  gc_DbmTranslation_fr_Text97 : WSTRING(28) := "White Light AVG actual value";
  gc_DbmTranslation_fr_Text98 : WSTRING(23) := "White Light AVD command";
  gc_DbmTranslation_fr_Text99 : WSTRING(28) := "White Light AVD actual value";
  gc_DbmTranslation_fr_Text100 : WSTRING(21) := "Red Light AVG command";
  gc_DbmTranslation_fr_Text101 : WSTRING(26) := "Red Light AVG actual value";
  gc_DbmTranslation_fr_Text102 : WSTRING(21) := "Red Light AVD command";
  gc_DbmTranslation_fr_Text103 : WSTRING(26) := "Red Light AVD actual value";
  gc_DbmTranslation_fr_Text104 : WSTRING(23) := "White Light ARG command";
  gc_DbmTranslation_fr_Text105 : WSTRING(28) := "White Light ARG actual value";
  gc_DbmTranslation_fr_Text106 : WSTRING(23) := "White Light ARD command";
  gc_DbmTranslation_fr_Text107 : WSTRING(28) := "White Light ARD actual value";
  gc_DbmTranslation_fr_Text108 : WSTRING(21) := "Red Light ARG command";
  gc_DbmTranslation_fr_Text109 : WSTRING(26) := "Red Light ARG actual value";
  gc_DbmTranslation_fr_Text110 : WSTRING(21) := "Red Light ARD command";
  gc_DbmTranslation_fr_Text111 : WSTRING(26) := "Red Light ARD actual value";
  gc_DbmTranslation_fr_Text112 : WSTRING(29) := "Suplly Pvg Left Track command";
  gc_DbmTranslation_fr_Text113 : WSTRING(34) := "Suplly Pvg Left Track actual value";
  gc_DbmTranslation_fr_Text114 : WSTRING(30) := "Suplly Pvg Right Track command";
  gc_DbmTranslation_fr_Text115 : WSTRING(35) := "Suplly Pvg Right Track actual value";
  gc_DbmTranslation_fr_Text116 : WSTRING(33) := "Ev UnBlock Oscillation Axle state";
  gc_DbmTranslation_fr_Text117 : WSTRING(40) := "Ev UnBlock Oscillation Axle command bool";
  gc_DbmTranslation_fr_Text118 : WSTRING(26) := "Ev Up Axle Oscillant state";
  gc_DbmTranslation_fr_Text119 : WSTRING(33) := "Ev Up Axle Oscillant Command Bool";
  gc_DbmTranslation_fr_Text120 : WSTRING(29) := "Ev Down Axle Oscillant  state";
  gc_DbmTranslation_fr_Text121 : WSTRING(35) := "Ev Down Axle Oscillant Command Bool";
  gc_DbmTranslation_fr_Text122 : WSTRING(20) := "Ev Up AxleFixe state";
  gc_DbmTranslation_fr_Text123 : WSTRING(28) := "Ev Up Axle Fixe Command Bool";
  gc_DbmTranslation_fr_Text124 : WSTRING(22) := "Ev Down AxleFixe state";
  gc_DbmTranslation_fr_Text125 : WSTRING(30) := "Ev Down Axle Fixe Command Bool";
  gc_DbmTranslation_fr_Text126 : WSTRING(35) := "Ev Park Brake Axle Oscillant  state";
  gc_DbmTranslation_fr_Text127 : WSTRING(42) := "Ev Park Brake Axle Oscillant  command bool";
  gc_DbmTranslation_fr_Text128 : WSTRING(29) := "Ev Park Brake Axle Fixe state";
  gc_DbmTranslation_fr_Text129 : WSTRING(37) := "Ev Park Brake Axle Fixe  command bool";
  gc_DbmTranslation_fr_Text130 : WSTRING(37) := "Ev Service Brake Axle Oscillant state";
  gc_DbmTranslation_fr_Text131 : WSTRING(36) := "Ev Service Brake Axle 1 command Bool";
  gc_DbmTranslation_fr_Text132 : WSTRING(32) := "Ev Service Brake Axle Fixe state";
  gc_DbmTranslation_fr_Text133 : WSTRING(36) := "Ev Service Brake Axle 2 command Bool";
  gc_DbmTranslation_fr_Text134 : WSTRING(19) := "Klaxon Neotec state";
  gc_DbmTranslation_fr_Text135 : WSTRING(26) := "Klaxon Neotec command bool";
  gc_DbmTranslation_fr_Text136 : WSTRING(18) := "Forward pump state";
  gc_DbmTranslation_fr_Text137 : WSTRING(21) := "Forward pump  command";
  gc_DbmTranslation_fr_Text138 : WSTRING(27) := "Forward pump actual current";
  gc_DbmTranslation_fr_Text139 : WSTRING(19) := "Backward pump state";
  gc_DbmTranslation_fr_Text140 : WSTRING(22) := "Backward pump  command";
  gc_DbmTranslation_fr_Text141 : WSTRING(28) := "Backward pump actual current";
  gc_DbmTranslation_fr_Text142 : WSTRING(22) := "Pvg left track command";
  gc_DbmTranslation_fr_Text143 : WSTRING(29) := "Pvg left track actual voltage";
  gc_DbmTranslation_fr_Text144 : WSTRING(23) := "Pvg right track command";
  gc_DbmTranslation_fr_Text145 : WSTRING(30) := "Pvg right track actual voltage";
  gc_DbmTranslation_fr_Text146 : WSTRING(26) := "Supply Ana Sensors Command";
  gc_DbmTranslation_fr_Text147 : WSTRING(24) := "Supply Ana Sensors Value";
  gc_DbmTranslation_fr_Text148 : WSTRING(30) := "Pvg Left Track Lowside Command";
  gc_DbmTranslation_fr_Text149 : WSTRING(28) := "Pvg Left Track Lowside Value";
  gc_DbmTranslation_fr_Text150 : WSTRING(31) := "Pvg Right Track Lowside Command";
  gc_DbmTranslation_fr_Text151 : WSTRING(29) := "Pvg Right Track Lowside Value";
  gc_DbmTranslation_fr_Text152 : WSTRING(39) := "Return low side Ev Forward Pump command";
  gc_DbmTranslation_fr_Text153 : WSTRING(37) := "Return low side Ev Forward Pump state";
  gc_DbmTranslation_fr_Text154 : WSTRING(40) := "Return low side Ev Backward Pump command";
  gc_DbmTranslation_fr_Text155 : WSTRING(38) := "Return low side Ev Backward Pump state";
  gc_DbmTranslation_fr_Text156 : WSTRING(19) := "Neon Lights command";
  gc_DbmTranslation_fr_Text157 : WSTRING(17) := "Neon Lights value";
  gc_DbmTranslation_fr_Text158 : WSTRING(33) := "Ev 2 Deflector Transmission value";
  gc_DbmTranslation_fr_Text159 : WSTRING(21) := "Cooling relay command";
  gc_DbmTranslation_fr_Text160 : WSTRING(19) := "Cooling relay state";
  gc_DbmTranslation_fr_Text161 : WSTRING(54) := "Sorties d’activation de l’Ev du deuxième frein de parc";
  gc_DbmTranslation_fr_Text162 : WSTRING(54) := "Sorties d’activation de l’Ev du deuxième frein de parc";
  gc_DbmTranslation_fr_Text163 : WSTRING(33) := "Ev 2nd Park Brake Axle Fixe State";
  gc_DbmTranslation_fr_Text164 : WSTRING(33) := "Ev 2nd Park Brake Axle Osci State";
  gc_DbmTranslation_fr_Text165 : WSTRING(41) := "Pvg Translation for Rail Electric Command";
  gc_DbmTranslation_fr_Text166 : WSTRING(41) := "Pvg Translation for Rail Electric Voltage";
  gc_DbmTranslation_fr_Text167 : WSTRING(48) := "Suplly Pvg Translation for Rail Electric Command";
  gc_DbmTranslation_fr_Text168 : WSTRING(46) := "Suplly Pvg Translation for Rail Electric State";
  gc_DbmTranslation_fr_Text169 : WSTRING(42) := "Ev Deviator for Rail Electric Mode Command";
  gc_DbmTranslation_fr_Text170 : WSTRING(40) := "Ev Deviator for Rail Electric Mode State";
  gc_DbmTranslation_fr_Text171 : WSTRING(43) := "Relay Cut Off Variator for Electric Command";
  gc_DbmTranslation_fr_Text172 : WSTRING(41) := "Relay Cut Off Variator for Electric State";
  gc_DbmTranslation_fr_Text173 : WSTRING(28) := "Relay Enable Battery Command";
  gc_DbmTranslation_fr_Text174 : WSTRING(26) := "Relay Enable Battery State";
  gc_DbmTranslation_fr_Text175 : WSTRING(25) := "Byte increased each cycle";
  gc_DbmTranslation_fr_Text176 : WSTRING(22) := "Watchdog current state";
  gc_DbmTranslation_fr_Text177 : WSTRING(11) := "Ecu voltage";
  gc_DbmTranslation_fr_Text178 : WSTRING(13) := "Off Rail Mode";
  gc_DbmTranslation_fr_Text179 : WSTRING(9) := "Rail Mode";
  gc_DbmTranslation_fr_Text180 : WSTRING(75) := "Output value Lut of Manipulator left radio control in range -10000 to 10000";
  gc_DbmTranslation_fr_Text181 : WSTRING(35) := "Output value Lut of Left Track Pvg ";
  gc_DbmTranslation_fr_Text182 : WSTRING(76) := "Output value Lut of Manipulator Right radio control in range -10000 to 10000";
  gc_DbmTranslation_fr_Text183 : WSTRING(36) := "Output value Lut of Right Track Pvg ";
  gc_DbmTranslation_fr_Text184 : WSTRING(52) := "Outût value Lut of Joystick advance Rail translation";
  gc_DbmTranslation_fr_Text185 : WSTRING(40) := "Output Lut  of Forward Pump Transmission";
  gc_DbmTranslation_fr_Text186 : WSTRING(41) := "Output Lut  of Backward Pump Transmission";
  gc_DbmTranslation_fr_Text187 : WSTRING(71) := "Calculate consigne current of Forward Pump transmission on percent *100";
  gc_DbmTranslation_fr_Text188 : WSTRING(24) := "LastJoystickAdvanceValue";
  gc_DbmTranslation_fr_Text189 : WSTRING(37) := "Scaling Value of Joystick advancement";
  gc_DbmTranslation_fr_Text190 : WSTRING(39) := "State of service brake rail translation";
  gc_DbmTranslation_fr_Text191 : WSTRING(36) := "Enable Start timer for service brake";
  gc_DbmTranslation_fr_Text192 : WSTRING(48) := "Speed motor command provide by track transaltion";
  gc_DbmTranslation_fr_Text193 : WSTRING(28) := "Force silent mode motor test";
  gc_DbmTranslation_fr_Text194 : WSTRING(19) := "Angular sensor test";
  gc_DbmTranslation_fr_Text195 : WSTRING(17) := "Speed axle sensor";
  gc_DbmTranslation_fr_Text196 : WSTRING(18) := "Average Time cycle";
  gc_DbmTranslation_fr_Text197 : WSTRING(14) := "Max time cycle";
  gc_DbmTranslation_fr_Text198 : WSTRING(40) := "First translation for release park brake";
  gc_DbmTranslation_fr_Text199 : WSTRING(35) := "Autorize Up Axle Oscillant movement";
  gc_DbmTranslation_fr_Text200 : WSTRING(37) := "Autorize Down Axle Oscillant movement";
  gc_DbmTranslation_fr_Text201 : WSTRING(30) := "Autorize Up Axle fixe movement";
  gc_DbmTranslation_fr_Text202 : WSTRING(32) := "Autorize Down Axle fixe movement";
  gc_DbmTranslation_fr_Text203 : WSTRING(19) := "Engine On run phase";
  gc_DbmTranslation_fr_Text204 : WSTRING(74) := "Transaltion rail or off rail is solicited , flag send to C1 to pilot motor";
  gc_DbmTranslation_fr_Text205 : WSTRING(42) := "Direction of rail translation (Av Ar Stop)";
  gc_DbmTranslation_fr_Text206 : WSTRING(39) := "Set condition to active Aru radio alarm";
  gc_DbmTranslation_fr_Text207 : WSTRING(36) := "Joystick advance setpoint after ramp";
  gc_DbmTranslation_fr_Text208 : WSTRING(46) := "Stabilized stop flag to active park brake rail";
  gc_DbmTranslation_fr_Text209 : WSTRING(48) := "Emergency brake flag to active sequence of brake";
  gc_DbmTranslation_fr_Text210 : WSTRING(51) := "Flag when the timer emergency service brake is done";
  gc_DbmTranslation_fr_Text211 : WSTRING(66) := "Flag when the timer stopped machine unblock osciilant axle is done";
  gc_DbmTranslation_fr_Text212 : WSTRING(86) := "Output value Lut of Manipulator left radio control in range -10000 to 10000 after ramp";
  gc_DbmTranslation_fr_Text213 : WSTRING(87) := "Output value Lut of Manipulator right radio control in range -10000 to 10000 after ramp";
  gc_DbmTranslation_fr_Text214 : WSTRING(52) := "Delta beetwen left and right Pvg crawler advancement";
  gc_DbmTranslation_fr_Text215 : WSTRING(65) := "Consigne left pvg track calcul with delta beetween left and right";
  gc_DbmTranslation_fr_Text216 : WSTRING(66) := "Consigne right pvg track calcul with delta beetween left and right";
  gc_DbmTranslation_fr_Text217 : WSTRING(56) := "Flag to detect brake when gachette or pedal are released";
  gc_DbmTranslation_fr_Text218 : WSTRING(50) := "Counter for debug when alarm aru radio is detected";
  gc_DbmTranslation_fr_Text219 : WSTRING(28) := "Red light ARG basket command";
  gc_DbmTranslation_fr_Text220 : WSTRING(30) := "White light ARG basket command";
  gc_DbmTranslation_fr_Text221 : WSTRING(32) := "Portilon close and ladder folded";
  gc_DbmTranslation_fr_Text222 : WSTRING(46) := "Test boolean  command to refresh objet evision";
  gc_DbmTranslation_fr_Text223 : WSTRING(60) := "Position of joysstick advancment ( AV_JOY, NEU_JOY , AR_JOY)";
  gc_DbmTranslation_fr_Text224 : WSTRING(81) := "Retain position of joystick advancement , reset when brake sequence is sollicited";
  gc_DbmTranslation_fr_Text225 : WSTRING(37) := "Authorize forward crawler translation";
  gc_DbmTranslation_fr_Text226 : WSTRING(38) := "Authorize backward crawler translation";
  gc_DbmTranslation_fr_Text227 : WSTRING(22) := "Return value uart init";
  gc_DbmTranslation_fr_Text228 : WSTRING(35) := "Authorize translation rail movement";
  gc_DbmTranslation_fr_Text229 : WSTRING(25) := "Ev forward track consigne";
  gc_DbmTranslation_fr_Text230 : WSTRING(24) := "Ev forward rail consigne";
  gc_DbmTranslation_fr_Text231 : WSTRING(0) := "";
  gc_DbmTranslation_fr_Text232 : WSTRING(21) := "Variable debug Neotec";
  gc_DbmTranslation_fr_Text233 : WSTRING(21) := "Variable debug Neotec";
  gc_DbmTranslation_fr_Text234 : WSTRING(21) := "Variable debug Neotec";
  gc_DbmTranslation_fr_Text235 : WSTRING(21) := "Variable debug Neotec";
  gc_DbmTranslation_fr_Text236 : WSTRING(21) := "Variable debug Neotec";
  gc_DbmTranslation_fr_Text237 : WSTRING(21) := "Variable debug Neotec";
  gc_DbmTranslation_fr_Text238 : WSTRING(21) := "Variable debug Neotec";
  gc_DbmTranslation_fr_Text239 : WSTRING(21) := "Variable debug Neotec";
  gc_DbmTranslation_fr_Text240 : WSTRING(21) := "Variable debug Neotec";
  gc_DbmTranslation_fr_Text241 : WSTRING(21) := "Variable debug Neotec";
  gc_DbmTranslation_fr_Text242 : WSTRING(21) := "Variable debug Neotec";
  gc_DbmTranslation_fr_Text243 : WSTRING(21) := "Variable debug Neotec";
  gc_DbmTranslation_fr_Text244 : WSTRING(21) := "Variable debug Neotec";
  gc_DbmTranslation_fr_Text245 : WSTRING(21) := "Variable debug Neotec";
  gc_DbmTranslation_fr_Text246 : WSTRING(21) := "Variable debug Neotec";
  gc_DbmTranslation_fr_Text247 : WSTRING(21) := "Variable debug Neotec";
  gc_DbmTranslation_fr_Text248 : WSTRING(21) := "Variable debug Neotec";
  gc_DbmTranslation_fr_Text249 : WSTRING(21) := "Variable debug Neotec";
  gc_DbmTranslation_fr_Text250 : WSTRING(21) := "Variable debug Neotec";
  gc_DbmTranslation_fr_Text251 : WSTRING(21) := "Variable debug Neotec";
  gc_DbmTranslation_fr_Text252 : WSTRING(21) := "Variable debug Neotec";
  gc_DbmTranslation_fr_Text253 : WSTRING(21) := "Variable debug Neotec";
  gc_DbmTranslation_fr_Text254 : WSTRING(21) := "Variable debug Neotec";
  gc_DbmTranslation_fr_Text255 : WSTRING(21) := "Variable debug Neotec";
  gc_DbmTranslation_fr_Text256 : WSTRING(21) := "Variable debug Neotec";
  gc_DbmTranslation_fr_Text257 : WSTRING(21) := "Variable debug Neotec";
  gc_DbmTranslation_fr_Text258 : WSTRING(21) := "Variable debug Neotec";
  gc_DbmTranslation_fr_Text259 : WSTRING(21) := "Variable debug Neotec";
  gc_DbmTranslation_fr_Text260 : WSTRING(21) := "Variable debug Neotec";
  gc_DbmTranslation_fr_Text261 : WSTRING(21) := "Variable debug Neotec";
  gc_DbmTranslation_fr_Text262 : WSTRING(21) := "Variable debug Neotec";
  gc_DbmTranslation_fr_Text263 : WSTRING(21) := "Variable debug Neotec";
  gc_DbmTranslation_fr_Text264 : WSTRING(21) := "Variable debug Neotec";
  gc_DbmTranslation_fr_Text265 : WSTRING(21) := "Variable debug Neotec";
  gc_DbmTranslation_fr_Text266 : WSTRING(21) := "Variable debug Neotec";
  gc_DbmTranslation_fr_Text267 : WSTRING(21) := "Variable debug Neotec";
  gc_DbmTranslation_fr_Text268 : WSTRING(21) := "Variable debug Neotec";
  gc_DbmTranslation_fr_Text269 : WSTRING(21) := "Variable debug Neotec";
  gc_DbmTranslation_fr_Text270 : WSTRING(21) := "Variable debug Neotec";
  gc_DbmTranslation_fr_Text271 : WSTRING(21) := "Variable debug Neotec";
  gc_DbmTranslation_fr_Text272 : WSTRING(28) := "Red light ARD basket command";
  gc_DbmTranslation_fr_Text273 : WSTRING(30) := "White light ARD basket command";
  gc_DbmTranslation_fr_Text274 : WSTRING(26) := "Active failure is detected";
  gc_DbmTranslation_fr_Text275 : WSTRING(19) := "Reduction pump rail";
  gc_DbmTranslation_fr_Text276 : WSTRING(20) := "Reduction pump track";
  gc_DbmTranslation_fr_Text277 : WSTRING(25) := "Active white lights 15746";
  gc_DbmTranslation_fr_Text278 : WSTRING(24) := "White light Av 15746 Cmd";
  gc_DbmTranslation_fr_Text279 : WSTRING(24) := "White light Ar 15746 Cmd";
  gc_DbmTranslation_fr_Text280 : WSTRING(38) := "Shunt all logic to test electricall IO";
  gc_DbmTranslation_fr_Text281 : WSTRING(29) := "Send Event Datalogger Message";
  gc_DbmTranslation_fr_Text282 : WSTRING(21) := "Depend de l’option MG";
  gc_DbmTranslation_fr_Text283 : WSTRING(13) := "Slow Blinking";
  gc_DbmTranslation_fr_Text284 : WSTRING(14) := "Total distance";
  gc_DbmTranslation_fr_Text285 : WSTRING(19) := "Running Stable 48XS";
  gc_DbmTranslation_fr_Text286 : WSTRING(39) := "Alarm Hydraulic Temperature Rail Active";
  gc_DbmTranslation_fr_Text287 : WSTRING(42) := "Alarm Hydraulic Temperature Crawler Active";
  gc_DbmTranslation_fr_Text288 : WSTRING(17) := "Diag Faulty Value";
  gc_DbmTranslation_fr_Text289 : WSTRING(15) := "Diag Device Num";
  gc_DbmTranslation_fr_Text290 : WSTRING(15) := "Diag Error Code";
  gc_DbmTranslation_fr_Text291 : WSTRING(21) := "Engine running stable";
  gc_DbmTranslation_fr_Text292 : WSTRING(42) := "Select config hollandaise to control light";
  gc_DbmTranslation_fr_Text293 : WSTRING(37) := "Portillon is installed on the machine";
  gc_DbmTranslation_fr_Text294 : WSTRING(34) := "Ladder is installed on the machine";
  gc_DbmTranslation_fr_Text295 : WSTRING(41) := "Measuring mat is installed on the machine";
  gc_DbmTranslation_fr_Text296 : WSTRING(107) := "-SpeedMaxRail Acces Site- Inclinaison Baslet most be in low sector for acces site speed on translation rail";
  gc_DbmTranslation_fr_Text297 : WSTRING(90) := "-SpeedMaxRail Acces Site- Basket most be centered for acces site speed on translation rail";
  gc_DbmTranslation_fr_Text298 : WSTRING(64) := "The digital display o the measuring mast is used on this vehicle";
  gc_DbmTranslation_fr_Text299 : WSTRING(30) := "Autorisation work key present ";
  gc_DbmTranslation_fr_Text300 : WSTRING(40) := "Option d’activation du mode double frein";
  gc_DbmTranslation_fr_Text301 : WSTRING(50) := "Strukton configuration for new performance machine";
  gc_DbmTranslation_fr_Text302 : WSTRING(46) := "Basket and turret limited by a mechanical stop";
  gc_DbmTranslation_fr_Text303 : WSTRING(24) := "Presence of sensor plate";
  gc_DbmTranslation_fr_Text304 : WSTRING(29) := "Number of brake cycle perform";
  gc_DbmTranslation_fr_Text305 : WSTRING(10) := "Light mode";
  gc_DbmTranslation_fr_Text306 : WSTRING(0) := "";
  gc_DbmTranslation_fr_Text307 : WSTRING(0) := "";
  gc_DbmTranslation_fr_Text308 : WSTRING(0) := "";
  gc_DbmTranslation_fr_Text309 : WSTRING(0) := "";
  gc_DbmTranslation_fr_Text310 : WSTRING(0) := "";
  gc_DbmTranslation_fr_Text311 : WSTRING(0) := "";
  gc_DbmTranslation_fr_Text312 : WSTRING(0) := "";
  gc_DbmTranslation_fr_Text313 : WSTRING(0) := "";
  gc_DbmTranslation_fr_Text314 : WSTRING(0) := "";
  gc_DbmTranslation_fr_Text315 : WSTRING(0) := "";
  gc_DbmTranslation_fr_Text316 : WSTRING(0) := "";
  gc_DbmTranslation_fr_Text317 : WSTRING(0) := "";
  gc_DbmTranslation_fr_Text318 : WSTRING(0) := "";
  gc_DbmTranslation_fr_Text319 : WSTRING(0) := "";
  gc_DbmTranslation_fr_Text320 : WSTRING(0) := "";
  gc_DbmTranslation_fr_Text321 : WSTRING(54) := "Nombres de cycle de frein pour les freins additionnels";
  gc_DbmTranslation_fr_Text322 : WSTRING(18) := "Total Distance Msb";
  gc_DbmTranslation_fr_Text323 : WSTRING(18) := "Total Distance Lsb";
  gc_DbmTranslation_fr_Text324 : WSTRING(77) := "Limit threshold of angle to stop movement , angular sensor from radio control";
  gc_DbmTranslation_fr_Text325 : WSTRING(43) := "Treshold minimal speed to active park brake";
  gc_DbmTranslation_fr_Text326 : WSTRING(46) := "Treshold minimal speed to active service brake";
  gc_DbmTranslation_fr_Text327 : WSTRING(41) := "Additionnal Pourcent Forward Pump Command";
  gc_DbmTranslation_fr_Text328 : WSTRING(67) := "Additionnal Pourcent Forward Pump Command when sient mode is active";
  gc_DbmTranslation_fr_Text329 : WSTRING(21) := "Node Id radio command";
  gc_DbmTranslation_fr_Text330 : WSTRING(34) := "Dead Zone joystick rotation turret";
  gc_DbmTranslation_fr_Text331 : WSTRING(52) := "Timer before 2nd Service Axle brake rail translation";
  gc_DbmTranslation_fr_Text332 : WSTRING(26) := "Time Service Brake Offrail";
  gc_DbmTranslation_fr_Text333 : WSTRING(59) := "Ev Forward Pump - PWM output parameters- engine off current";
  gc_DbmTranslation_fr_Text334 : WSTRING(56) := "Ev Forward Pump - PWM output parameters- minimal current";
  gc_DbmTranslation_fr_Text335 : WSTRING(54) := "Ev Forward Pump - PWM output parameters- stop current ";
  gc_DbmTranslation_fr_Text336 : WSTRING(60) := "Ev Backward Pump - PWM output parameters- engine off current";
  gc_DbmTranslation_fr_Text337 : WSTRING(57) := "Ev Backward Pump - PWM output parameters- minimal current";
  gc_DbmTranslation_fr_Text338 : WSTRING(55) := "Ev Backward Pump - PWM output parameters- stop current ";
  gc_DbmTranslation_fr_Text339 : WSTRING(67) := "Position neutral of joystick advancement regarding batterie voltage";
  gc_DbmTranslation_fr_Text340 : WSTRING(46) := "PID - Ev Forward Pump - Gp - proportional gain";
  gc_DbmTranslation_fr_Text341 : WSTRING(54) := "PID - Ev Forward Pump - Ti - integration time constant";
  gc_DbmTranslation_fr_Text342 : WSTRING(53) := "PID - Ev Forward Pump - Td - derivation time constant";
  gc_DbmTranslation_fr_Text343 : WSTRING(46) := "PID - Ev Forward Pump - Gp - proportional gain";
  gc_DbmTranslation_fr_Text344 : WSTRING(54) := "PID - Ev Forward Pump - Ti - integration time constant";
  gc_DbmTranslation_fr_Text345 : WSTRING(53) := "PID - Ev Forward Pump - Td - derivation time constant";
  gc_DbmTranslation_fr_Text346 : WSTRING(80) := "PressureBlockOscillationSensor - input current - output characteristic - Positif";
  gc_DbmTranslation_fr_Text347 : WSTRING(80) := "PressureBlockOscillationSensor - input current - output characteristic - Neutral";
  gc_DbmTranslation_fr_Text348 : WSTRING(80) := "PressureBlockOscillationSensor - input current - output characteristic - Negatif";
  gc_DbmTranslation_fr_Text349 : WSTRING(69) := "PressureBrakeSensor - input current - output characteristic - Positif";
  gc_DbmTranslation_fr_Text350 : WSTRING(69) := "PressureBrakeSensor - input current - output characteristic - Neutral";
  gc_DbmTranslation_fr_Text351 : WSTRING(69) := "PressureBrakeSensor - input current - output characteristic - Negatif";
  gc_DbmTranslation_fr_Text352 : WSTRING(79) := "TemperatureTransmissionSensor - input current - output characteristic - Positif";
  gc_DbmTranslation_fr_Text353 : WSTRING(79) := "TemperatureTransmissionSensor - input current - output characteristic - Neutral";
  gc_DbmTranslation_fr_Text354 : WSTRING(79) := "TemperatureTransmissionSensor - input current - output characteristic - Negatif";
  gc_DbmTranslation_fr_Text355 : WSTRING(55) := "Consigne min Ev forward apply with joystick advancement";
  gc_DbmTranslation_fr_Text356 : WSTRING(55) := "Consigne max Ev forward apply with joystick advancement";
  gc_DbmTranslation_fr_Text357 : WSTRING(56) := "Consigne min Ev backward apply with joystick advancement";
  gc_DbmTranslation_fr_Text358 : WSTRING(56) := "Consigne max Ev backward apply with joystick advancement";
  gc_DbmTranslation_fr_Text359 : WSTRING(96) := "Time  ramp to Ev rail [0] Pos incr time, [1] Pos decr time,[2] Neg incr time , [3] Neg decr time";
  gc_DbmTranslation_fr_Text360 : WSTRING(96) := "Time  ramp to Ev rail [0] Pos incr time, [1] Pos decr time,[2] Neg incr time , [3] Neg decr time";
  gc_DbmTranslation_fr_Text361 : WSTRING(96) := "Time  ramp to Ev rail [0] Pos incr time, [1] Pos decr time,[2] Neg incr time , [3] Neg decr time";
  gc_DbmTranslation_fr_Text362 : WSTRING(96) := "Time  ramp to Ev rail [0] Pos incr time, [1] Pos decr time,[2] Neg incr time , [3] Neg decr time";
  gc_DbmTranslation_fr_Text363 : WSTRING(96) := "Time  ramp to Ev rail [0] Pos incr time, [1] Pos decr time,[2] Neg incr time , [3] Neg decr time";
  gc_DbmTranslation_fr_Text364 : WSTRING(53) := "Consigne min Ev forward apply for crawler advancement";
  gc_DbmTranslation_fr_Text365 : WSTRING(53) := "Consigne max Ev forward apply for crawler advancement";
  gc_DbmTranslation_fr_Text366 : WSTRING(72) := "Ratio apply to ramp signal to control Ev forward for crawler advancement";
  gc_DbmTranslation_fr_Text367 : WSTRING(72) := "Ratio apply to ramp signal to control Ev forward for crawler advancement";
  gc_DbmTranslation_fr_Text368 : WSTRING(72) := "Ratio apply to ramp signal to control Ev forward for crawler advancement";
  gc_DbmTranslation_fr_Text369 : WSTRING(69) := "Park Brake rail - Treshold of regime motor to active park brake rail ";
  gc_DbmTranslation_fr_Text370 : WSTRING(95) := "Consigne min Pvg Left Track apply when mapinulator get out neutral position to forward position";
  gc_DbmTranslation_fr_Text371 : WSTRING(30) := "Consigne max Pvg Left Track Av";
  gc_DbmTranslation_fr_Text372 : WSTRING(96) := "Consigne min Pvg Left Track apply when mapinulator get out neutral position to backward position";
  gc_DbmTranslation_fr_Text373 : WSTRING(30) := "Consigne max Pvg Left Track Ar";
  gc_DbmTranslation_fr_Text374 : WSTRING(96) := "Consigne min Pvg Right Track apply when mapinulator get out neutral position to forward position";
  gc_DbmTranslation_fr_Text375 : WSTRING(31) := "Consigne max Pvg Right Track Av";
  gc_DbmTranslation_fr_Text376 : WSTRING(97) := "Consigne min Pvg Right Track apply when mapinulator get out neutral position to backward position";
  gc_DbmTranslation_fr_Text377 : WSTRING(31) := "Consigne max Pvg Right Track Ar";
  gc_DbmTranslation_fr_Text378 : WSTRING(105) := "Time  ramp apply to left track [0] Pos incr time, [1] Pos decr time,[2] Neg incr time , [3] Neg decr time";
  gc_DbmTranslation_fr_Text379 : WSTRING(105) := "Time  ramp apply to left track [0] Pos incr time, [1] Pos decr time,[2] Neg incr time , [3] Neg decr time";
  gc_DbmTranslation_fr_Text380 : WSTRING(105) := "Time  ramp apply to left track [0] Pos incr time, [1] Pos decr time,[2] Neg incr time , [3] Neg decr time";
  gc_DbmTranslation_fr_Text381 : WSTRING(105) := "Time  ramp apply to left track [0] Pos incr time, [1] Pos decr time,[2] Neg incr time , [3] Neg decr time";
  gc_DbmTranslation_fr_Text382 : WSTRING(105) := "Time  ramp apply to left track [0] Pos incr time, [1] Pos decr time,[2] Neg incr time , [3] Neg decr time";
  gc_DbmTranslation_fr_Text383 : WSTRING(106) := "Time  ramp apply to right track [0] Pos incr time, [1] Pos decr time,[2] Neg incr time , [3] Neg decr time";
  gc_DbmTranslation_fr_Text384 : WSTRING(106) := "Time  ramp apply to right track [0] Pos incr time, [1] Pos decr time,[2] Neg incr time , [3] Neg decr time";
  gc_DbmTranslation_fr_Text385 : WSTRING(106) := "Time  ramp apply to right track [0] Pos incr time, [1] Pos decr time,[2] Neg incr time , [3] Neg decr time";
  gc_DbmTranslation_fr_Text386 : WSTRING(106) := "Time  ramp apply to right track [0] Pos incr time, [1] Pos decr time,[2] Neg incr time , [3] Neg decr time";
  gc_DbmTranslation_fr_Text387 : WSTRING(106) := "Time  ramp apply to right track [0] Pos incr time, [1] Pos decr time,[2] Neg incr time , [3] Neg decr time";
  gc_DbmTranslation_fr_Text388 : WSTRING(38) := "Time to detect stabilized stop machine";
  gc_DbmTranslation_fr_Text389 : WSTRING(67) := "Treshold low spped to start timer to detect stabilized stop machine";
  gc_DbmTranslation_fr_Text390 : WSTRING(66) := "Time before release service brake when emergency brake is detected";
  gc_DbmTranslation_fr_Text391 : WSTRING(57) := "Time stopped machine to controle unblock oscillation axle";
  gc_DbmTranslation_fr_Text392 : WSTRING(87) := "Low treshold speed of oscillation and fixe axle to start timer unblock oscillation axle";
  gc_DbmTranslation_fr_Text393 : WSTRING(55) := "Gap max beetween left and right Pvg crawler advancement";
  gc_DbmTranslation_fr_Text394 : WSTRING(84) := "Gap max beetween left and right Pvg crawler advancement when manipulator is inverted";
  gc_DbmTranslation_fr_Text395 : WSTRING(36) := "Treshold Ana to bool input from 48xs";
  gc_DbmTranslation_fr_Text396 : WSTRING(65) := "In min joystick advancement pourcentent by 10 of batterie voltage";
  gc_DbmTranslation_fr_Text397 : WSTRING(65) := "In max joystick advancement pourcentent by 10 of batterie voltage";
  gc_DbmTranslation_fr_Text398 : WSTRING(35) := "Speed mini treshol to re authorise ";
  gc_DbmTranslation_fr_Text399 : WSTRING(44) := "Number element for average slope trans angle";
  gc_DbmTranslation_fr_Text400 : WSTRING(43) := "Number element for average slope long angle";
  gc_DbmTranslation_fr_Text401 : WSTRING(35) := "Dead zone joystick rail advancement";
  gc_DbmTranslation_fr_Text402 : WSTRING(57) := "Number element for average slope trans angle 2nd channels";
  gc_DbmTranslation_fr_Text403 : WSTRING(56) := "Number element for average slope long angle 2nd channels";
  gc_DbmTranslation_fr_Text404 : WSTRING(18) := "Param debug Neotec";
  gc_DbmTranslation_fr_Text405 : WSTRING(18) := "Param debug Neotec";
  gc_DbmTranslation_fr_Text406 : WSTRING(18) := "Param debug Neotec";
  gc_DbmTranslation_fr_Text407 : WSTRING(18) := "Param debug Neotec";
  gc_DbmTranslation_fr_Text408 : WSTRING(18) := "Param debug Neotec";
  gc_DbmTranslation_fr_Text409 : WSTRING(18) := "Param debug Neotec";
  gc_DbmTranslation_fr_Text410 : WSTRING(18) := "Param debug Neotec";
  gc_DbmTranslation_fr_Text411 : WSTRING(18) := "Param debug Neotec";
  gc_DbmTranslation_fr_Text412 : WSTRING(18) := "Param debug Neotec";
  gc_DbmTranslation_fr_Text413 : WSTRING(18) := "Param debug Neotec";
  gc_DbmTranslation_fr_Text414 : WSTRING(18) := "Param debug Neotec";
  gc_DbmTranslation_fr_Text415 : WSTRING(18) := "Param debug Neotec";
  gc_DbmTranslation_fr_Text416 : WSTRING(18) := "Param debug Neotec";
  gc_DbmTranslation_fr_Text417 : WSTRING(18) := "Param debug Neotec";
  gc_DbmTranslation_fr_Text418 : WSTRING(18) := "Param debug Neotec";
  gc_DbmTranslation_fr_Text419 : WSTRING(18) := "Param debug Neotec";
  gc_DbmTranslation_fr_Text420 : WSTRING(18) := "Param debug Neotec";
  gc_DbmTranslation_fr_Text421 : WSTRING(57) := "Treshold hydraulique temperature to control cooling relay";
  gc_DbmTranslation_fr_Text422 : WSTRING(22) := "Time to control cooler";
  gc_DbmTranslation_fr_Text423 : WSTRING(37) := "Time fault pressure reduction crawler";
  gc_DbmTranslation_fr_Text424 : WSTRING(35) := "Rail joystick ratio two speed fault";
  gc_DbmTranslation_fr_Text425 : WSTRING(25) := "Timeout sdo resquest time";
  gc_DbmTranslation_fr_Text426 : WSTRING(29) := "Period Blinck off White Light";
  gc_DbmTranslation_fr_Text427 : WSTRING(48) := "filtrage et le lissage de la valeur du joystick.";
  gc_DbmTranslation_fr_Text428 : WSTRING(92) := "temporisation de l’AU afin d’attendre la fin des rampes avec un freinage d’urgence (Mode MG)";
  gc_DbmTranslation_fr_Text429 : WSTRING(59) := "seuil d’angle tourelle pour la petite vitesse, côté positif";
  gc_DbmTranslation_fr_Text430 : WSTRING(59) := "seuil d’angle tourelle pour la petite vitesse, côté négatif";
  gc_DbmTranslation_fr_Text431 : WSTRING(25) := "Number of file parameters";
  gc_DbmTranslation_fr_Text432 : WSTRING(13) := "Version Major";
  gc_DbmTranslation_fr_Text433 : WSTRING(14) := "Version Minior";
  gc_DbmTranslation_fr_Text434 : WSTRING(13) := "Version Patch";
  gc_DbmTranslation_fr_Text435 : WSTRING(14) := "Version Custom";
  gc_DbmTranslation_fr_Text436 : WSTRING(76) := "ElectricPumpPressureSensor - input current - output characteristic - Positif";
  gc_DbmTranslation_fr_Text437 : WSTRING(76) := "ElectricPumpPressureSensor - input current - output characteristic - Neutral";
  gc_DbmTranslation_fr_Text438 : WSTRING(76) := "ElectricPumpPressureSensor - input current - output characteristic - Negatif";
  gc_DbmTranslation_fr_Text439 : WSTRING(44) := "Max point Lut Manipulator Left radio control";
  gc_DbmTranslation_fr_Text440 : WSTRING(52) := "Lut array X value for Manipulator Left radio control";
  gc_DbmTranslation_fr_Text441 : WSTRING(52) := "Lut array X value for Manipulator Left radio control";
  gc_DbmTranslation_fr_Text442 : WSTRING(52) := "Lut array X value for Manipulator Left radio control";
  gc_DbmTranslation_fr_Text443 : WSTRING(52) := "Lut array Y value for Manipulator Left radio control";
  gc_DbmTranslation_fr_Text444 : WSTRING(52) := "Lut array Y value for Manipulator Left radio control";
  gc_DbmTranslation_fr_Text445 : WSTRING(52) := "Lut array Y value for Manipulator Left radio control";
  gc_DbmTranslation_fr_Text446 : WSTRING(45) := "Max point Lut Manipulator Right radio control";
  gc_DbmTranslation_fr_Text447 : WSTRING(53) := "Lut array X value for Manipulator Right radio control";
  gc_DbmTranslation_fr_Text448 : WSTRING(53) := "Lut array X value for Manipulator Right radio control";
  gc_DbmTranslation_fr_Text449 : WSTRING(53) := "Lut array X value for Manipulator Right radio control";
  gc_DbmTranslation_fr_Text450 : WSTRING(53) := "Lut array Y value for Manipulator Right radio control";
  gc_DbmTranslation_fr_Text451 : WSTRING(53) := "Lut array Y value for Manipulator Right radio control";
  gc_DbmTranslation_fr_Text452 : WSTRING(53) := "Lut array Y value for Manipulator Right radio control";
  gc_DbmTranslation_fr_Text453 : WSTRING(40) := "Max point Lut for Left track pvg command";
  gc_DbmTranslation_fr_Text454 : WSTRING(25) := "Left track Pvg Ramp ratio";
  gc_DbmTranslation_fr_Text455 : WSTRING(25) := "Left track Pvg Ramp ratio";
  gc_DbmTranslation_fr_Text456 : WSTRING(25) := "Left track Pvg Ramp ratio";
  gc_DbmTranslation_fr_Text457 : WSTRING(50) := "Range value of left track Pvg apply to ramp signal";
  gc_DbmTranslation_fr_Text458 : WSTRING(50) := "Range value of left track Pvg apply to ramp signal";
  gc_DbmTranslation_fr_Text459 : WSTRING(50) := "Range value of left track Pvg apply to ramp signal";
  gc_DbmTranslation_fr_Text460 : WSTRING(50) := "Range value of left track Pvg apply to ramp signal";
  gc_DbmTranslation_fr_Text461 : WSTRING(26) := "Right track Pvg Ramp ratio";
  gc_DbmTranslation_fr_Text462 : WSTRING(26) := "Right track Pvg Ramp ratio";
  gc_DbmTranslation_fr_Text463 : WSTRING(26) := "Right track Pvg Ramp ratio";
  gc_DbmTranslation_fr_Text464 : WSTRING(51) := "Range value of right track Pvg apply to ramp signal";
  gc_DbmTranslation_fr_Text465 : WSTRING(51) := "Range value of right track Pvg apply to ramp signal";
  gc_DbmTranslation_fr_Text466 : WSTRING(51) := "Range value of right track Pvg apply to ramp signal";
  gc_DbmTranslation_fr_Text467 : WSTRING(51) := "Range value of right track Pvg apply to ramp signal";
  gc_DbmTranslation_fr_Text468 : WSTRING(56) := "Max point Lut Forward pump transmission rail translation";
  gc_DbmTranslation_fr_Text469 : WSTRING(64) := "Lut array X value for Forward pump transmission rail translation";
  gc_DbmTranslation_fr_Text470 : WSTRING(64) := "Lut array X value for Forward pump transmission rail translation";
  gc_DbmTranslation_fr_Text471 : WSTRING(64) := "Lut array X value for Forward pump transmission rail translation";
  gc_DbmTranslation_fr_Text472 : WSTRING(64) := "Lut array Y value for Forward pump transmission rail translation";
  gc_DbmTranslation_fr_Text473 : WSTRING(64) := "Lut array Y value for Forward pump transmission rail translation";
  gc_DbmTranslation_fr_Text474 : WSTRING(64) := "Lut array Y value for Forward pump transmission rail translation";
  gc_DbmTranslation_fr_Text475 : WSTRING(57) := "Max point Lut Backward pump transmission rail translation";
  gc_DbmTranslation_fr_Text476 : WSTRING(64) := "Lut array X value for Backwardpump transmission rail translation";
  gc_DbmTranslation_fr_Text477 : WSTRING(64) := "Lut array X value for Backwardpump transmission rail translation";
  gc_DbmTranslation_fr_Text478 : WSTRING(64) := "Lut array X value for Backwardpump transmission rail translation";
  gc_DbmTranslation_fr_Text479 : WSTRING(64) := "Lut array Y value for Backwardpump transmission rail translation";
  gc_DbmTranslation_fr_Text480 : WSTRING(64) := "Lut array Y value for Backwardpump transmission rail translation";
  gc_DbmTranslation_fr_Text481 : WSTRING(64) := "Lut array Y value for Backwardpump transmission rail translation";
  gc_DbmTranslation_fr_Text482 : WSTRING(36) := "Forward pump transmission Ramp ratio";
  gc_DbmTranslation_fr_Text483 : WSTRING(36) := "Forward pump transmission Ramp ratio";
  gc_DbmTranslation_fr_Text484 : WSTRING(36) := "Forward pump transmission Ramp ratio";
  gc_DbmTranslation_fr_Text485 : WSTRING(51) := "Range value of Forward pump transmission Ramp ratio";
  gc_DbmTranslation_fr_Text486 : WSTRING(51) := "Range value of Forward pump transmission Ramp ratio";
  gc_DbmTranslation_fr_Text487 : WSTRING(51) := "Range value of Forward pump transmission Ramp ratio";
  gc_DbmTranslation_fr_Text488 : WSTRING(51) := "Range value of Forward pump transmission Ramp ratio";
  gc_DbmTranslation_fr_Text489 : WSTRING(37) := "Backward pump transmission Ramp ratio";
  gc_DbmTranslation_fr_Text490 : WSTRING(37) := "Backward pump transmission Ramp ratio";
  gc_DbmTranslation_fr_Text491 : WSTRING(37) := "Backward pump transmission Ramp ratio";
  gc_DbmTranslation_fr_Text492 : WSTRING(52) := "Range value of Backward pump transmission Ramp ratio";
  gc_DbmTranslation_fr_Text493 : WSTRING(52) := "Range value of Backward pump transmission Ramp ratio";
  gc_DbmTranslation_fr_Text494 : WSTRING(52) := "Range value of Backward pump transmission Ramp ratio";
  gc_DbmTranslation_fr_Text495 : WSTRING(52) := "Range value of Backward pump transmission Ramp ratio";
  gc_DbmTranslation_fr_Text496 : WSTRING(38) := "Offset apply to calcul angle of turret";
  gc_DbmTranslation_fr_Text497 : WSTRING(55) := "Slope Long offset to calibrate value of longetude angle";
  gc_DbmTranslation_fr_Text498 : WSTRING(58) := "Slope Trans offset to calibrate value of transversal angle";
  gc_DbmTranslation_fr_Text499 : WSTRING(68) := "Slope Long offset to calibrate value of longetude angle 2nd channels";
  gc_DbmTranslation_fr_Text500 : WSTRING(71) := "Slope Trans offset to calibrate value of transversal angle 2nd channels";
  gc_DbmTranslation_fr_Text501 : WSTRING(53) := "Offset apply to calcul angle of turret second channel";
  gc_DbmTranslation_fr_Text502 : WSTRING(21) := "Encodeur Turret Msb 1";
  gc_DbmTranslation_fr_Text503 : WSTRING(21) := "Encodeur Turret Msb 2";
  gc_DbmTranslation_fr_Text504 : WSTRING(21) := "Encodeur Turret Lsb 1";
  gc_DbmTranslation_fr_Text505 : WSTRING(21) := "Encodeur Turret Lsb 2";
  gc_DbmTranslation_fr_Text506 : WSTRING(29) := "Up  Inclinaison basket button";
  gc_DbmTranslation_fr_Text507 : WSTRING(40) := "Up  Inclinaison basket  button raw value";
  gc_DbmTranslation_fr_Text508 : WSTRING(31) := "Down  Inclinaison basket button";
  gc_DbmTranslation_fr_Text509 : WSTRING(41) := "Down  Inclinaison basket button raw value";
  gc_DbmTranslation_fr_Text510 : WSTRING(18) := "Up pendular button";
  gc_DbmTranslation_fr_Text511 : WSTRING(28) := "Up pendular button raw value";
  gc_DbmTranslation_fr_Text512 : WSTRING(20) := "Down pendular button";
  gc_DbmTranslation_fr_Text513 : WSTRING(30) := "Down pendular button raw value";
  gc_DbmTranslation_fr_Text514 : WSTRING(40) := "Counter Clockwise rotation basket button";
  gc_DbmTranslation_fr_Text515 : WSTRING(50) := "Counter Clockwise rotation basket button raw value";
  gc_DbmTranslation_fr_Text516 : WSTRING(32) := "Clockwise rotation basket button";
  gc_DbmTranslation_fr_Text517 : WSTRING(42) := "Clockwise rotation basket button raw value";
  gc_DbmTranslation_fr_Text518 : WSTRING(10) := "Overload 1";
  gc_DbmTranslation_fr_Text519 : WSTRING(20) := "Overload 1 raw value";
  gc_DbmTranslation_fr_Text520 : WSTRING(10) := "Overload 2";
  gc_DbmTranslation_fr_Text521 : WSTRING(20) := "Overload 2 raw value";
  gc_DbmTranslation_fr_Text522 : WSTRING(34) := "Nacelle basket right side sensor 1";
  gc_DbmTranslation_fr_Text523 : WSTRING(40) := "Nacelle basket right side sensor 1 value";
  gc_DbmTranslation_fr_Text524 : WSTRING(35) := "Nacelle basket right side sensor 2 ";
  gc_DbmTranslation_fr_Text525 : WSTRING(40) := "Nacelle basket right side sensor 2 value";
  gc_DbmTranslation_fr_Text526 : WSTRING(33) := "Nacelle basket left side sensor 1";
  gc_DbmTranslation_fr_Text527 : WSTRING(39) := "Nacelle basket left side sensor 1 value";
  gc_DbmTranslation_fr_Text528 : WSTRING(33) := "Nacelle basket left side sensor 2";
  gc_DbmTranslation_fr_Text529 : WSTRING(39) := "Nacelle basket left side sensor 2 value";
  gc_DbmTranslation_fr_Text530 : WSTRING(26) := "Low sector pendular sensor";
  gc_DbmTranslation_fr_Text531 : WSTRING(32) := "Low sector pendular sensor value";
  gc_DbmTranslation_fr_Text532 : WSTRING(24) := "High Sector Plate Sensor";
  gc_DbmTranslation_fr_Text533 : WSTRING(30) := "High Sector Plate Sensor value";
  gc_DbmTranslation_fr_Text534 : WSTRING(20) := "Folded ladder sensor";
  gc_DbmTranslation_fr_Text535 : WSTRING(26) := "Folded ladder sensor value";
  gc_DbmTranslation_fr_Text536 : WSTRING(23) := "Safety man system value";
  gc_DbmTranslation_fr_Text537 : WSTRING(29) := "Delta arm axis joystick value";
  gc_DbmTranslation_fr_Text538 : WSTRING(29) := "Arrow arm axis joystick value";
  gc_DbmTranslation_fr_Text539 : WSTRING(33) := "Telescope arm axis joystick value";
  gc_DbmTranslation_fr_Text540 : WSTRING(35) := "Rotation turret axis joystick value";
  gc_DbmTranslation_fr_Text541 : WSTRING(27) := "Advance axis joystick value";
  gc_DbmTranslation_fr_Text542 : WSTRING(28) := "Rearmement Safety Man System";
  gc_DbmTranslation_fr_Text543 : WSTRING(34) := "Rearmement Safety Man System value";
  gc_DbmTranslation_fr_Text544 : WSTRING(28) := "Abutement Nacelle Track Side";
  gc_DbmTranslation_fr_Text545 : WSTRING(34) := "Abutement Nacelle Track Side value";
  gc_DbmTranslation_fr_Text546 : WSTRING(31) := "Abutement Nacelle Centered Side";
  gc_DbmTranslation_fr_Text547 : WSTRING(37) := "Abutement Nacelle Centered Side value";
  gc_DbmTranslation_fr_Text548 : WSTRING(24) := "Delta arm Joystick value";
  gc_DbmTranslation_fr_Text549 : WSTRING(38) := "Arrow Joystick / centered turret value";
  gc_DbmTranslation_fr_Text550 : WSTRING(31) := "Centered advance joystick value";
  gc_DbmTranslation_fr_Text551 : WSTRING(20) := "Dead man pedal value";
  gc_DbmTranslation_fr_Text552 : WSTRING(35) := "Pressence in nacelle sensor 1 value";
  gc_DbmTranslation_fr_Text553 : WSTRING(35) := "Pressence in nacelle sensor 2 value";
  gc_DbmTranslation_fr_Text554 : WSTRING(14) := "Gachette value";
  gc_DbmTranslation_fr_Text555 : WSTRING(12) := "Klaxon value";
  gc_DbmTranslation_fr_Text556 : WSTRING(17) := "Stop Motor button";
  gc_DbmTranslation_fr_Text557 : WSTRING(28) := "Authorization work key value";
  gc_DbmTranslation_fr_Text558 : WSTRING(27) := "Etallonnage Joystick Button";
  gc_DbmTranslation_fr_Text559 : WSTRING(22) := "Close Portillon Sensor";
  gc_DbmTranslation_fr_Text560 : WSTRING(31) := "Heartbeat for slave module 48xs";
  gc_DbmTranslation_fr_Text561 : WSTRING(37) := "Batterie voltage of module slave 48xs";
  gc_DbmTranslation_fr_Text562 : WSTRING(20) := "White Lights command";
  gc_DbmTranslation_fr_Text563 : WSTRING(25) := "White Lights actual value";
  gc_DbmTranslation_fr_Text564 : WSTRING(18) := "Red Lights command";
  gc_DbmTranslation_fr_Text565 : WSTRING(23) := "Red Lights actual value";
  gc_DbmTranslation_fr_Text566 : WSTRING(18) := "Work Light command";
  gc_DbmTranslation_fr_Text567 : WSTRING(18) := "Work Light command";
  gc_DbmTranslation_fr_Text568 : WSTRING(14) := "Buzzer command";
  gc_DbmTranslation_fr_Text569 : WSTRING(19) := "Buzzer actual value";
  gc_DbmTranslation_fr_Text570 : WSTRING(41) := "Error status of Motor Default Light ouput";
  gc_DbmTranslation_fr_Text571 : WSTRING(36) := "Error status of Overload Light ouput";
  gc_DbmTranslation_fr_Text572 : WSTRING(28) := "Error status of Buzzer ouput";
  gc_DbmTranslation_fr_Text573 : WSTRING(35) := "Error status of Gas Oil Light ouput";
  gc_DbmTranslation_fr_Text574 : WSTRING(42) := "Error status of devers default light ouput";
  gc_DbmTranslation_fr_Text575 : WSTRING(35) := "Error status of Red Light ARD ouput";
  gc_DbmTranslation_fr_Text576 : WSTRING(43) := "Error status of White Light ARD light ouput";
  gc_DbmTranslation_fr_Text577 : WSTRING(35) := "Error status of Warming Light ouput";
  gc_DbmTranslation_fr_Text578 : WSTRING(35) := "Error status of Red Light ARG ouput";
  gc_DbmTranslation_fr_Text579 : WSTRING(43) := "Error status of White Light ARG light ouput";
  gc_DbmTranslation_fr_Text580 : WSTRING(22) := "State of radio control";
  gc_DbmTranslation_fr_Text581 : WSTRING(16) := "Left manipulator";
  gc_DbmTranslation_fr_Text582 : WSTRING(17) := "Right manipulator";
  gc_DbmTranslation_fr_Text583 : WSTRING(23) := "LeftManipulatorPosition";
  gc_DbmTranslation_fr_Text584 : WSTRING(24) := "RightManipulatorPosition";
  gc_DbmTranslation_fr_Text585 : WSTRING(12) := "UpAxleArFixe";
  gc_DbmTranslation_fr_Text586 : WSTRING(14) := "DownAxleArFixe";
  gc_DbmTranslation_fr_Text587 : WSTRING(17) := "UpAxleAvOscillant";
  gc_DbmTranslation_fr_Text588 : WSTRING(19) := "DownAxleAvOscillant";
  gc_DbmTranslation_fr_Text589 : WSTRING(32) := "Rotation frame Coutner clockwise";
  gc_DbmTranslation_fr_Text590 : WSTRING(24) := "Rotation frame clockwise";
  gc_DbmTranslation_fr_Text591 : WSTRING(24) := "Selector rotation turret";
  gc_DbmTranslation_fr_Text592 : WSTRING(17) := "Selector pendular";
  gc_DbmTranslation_fr_Text593 : WSTRING(21) := "Radio command connect";
  gc_DbmTranslation_fr_Text594 : WSTRING(40) := "Up pendular or rotation clockwise turret";
  gc_DbmTranslation_fr_Text595 : WSTRING(50) := "down pendular or rotation counter clockwise turret";
  gc_DbmTranslation_fr_Text596 : WSTRING(19) := "Start radio command";
  gc_DbmTranslation_fr_Text597 : WSTRING(18) := "Stop radio command";
  gc_DbmTranslation_fr_Text598 : WSTRING(21) := "Forcing advance track";
  gc_DbmTranslation_fr_Text599 : WSTRING(14) := "Klaxon command";
  gc_DbmTranslation_fr_Text600 : WSTRING(27) := "Encodeur turret 1 angle raw";
  gc_DbmTranslation_fr_Text601 : WSTRING(51) := "Encodeur turret 1 angle with calibration parameters";
  gc_DbmTranslation_fr_Text602 : WSTRING(27) := "Encodeur turret 2 angle raw";
  gc_DbmTranslation_fr_Text603 : WSTRING(51) := "Encodeur turret 2 angle with calibration parameters";
  gc_DbmTranslation_fr_Text604 : WSTRING(26) := "Devers1 X axis angle value";
  gc_DbmTranslation_fr_Text605 : WSTRING(26) := "Devers1 Y axis angle value";
  gc_DbmTranslation_fr_Text606 : WSTRING(46) := "Slope Long Angle value with calibration offset";
  gc_DbmTranslation_fr_Text607 : WSTRING(47) := "Slope Trans Angle value with calibration offset";
  gc_DbmTranslation_fr_Text608 : WSTRING(30) := "State heart beat devers sensor";
  gc_DbmTranslation_fr_Text609 : WSTRING(41) := "State heart beat encodeur turret sensor 1";
  gc_DbmTranslation_fr_Text610 : WSTRING(20) := "Selected slope angle";
  gc_DbmTranslation_fr_Text611 : WSTRING(31) := "Encodeur mast measure raw value";
  gc_DbmTranslation_fr_Text612 : WSTRING(62) := "Encodeur mast measure with calibration parameters in centilmer";
  gc_DbmTranslation_fr_Text613 : WSTRING(26) := "Devers2 X axis angle value";
  gc_DbmTranslation_fr_Text614 : WSTRING(26) := "Devers2 Y axis angle value";
  gc_DbmTranslation_fr_Text615 : WSTRING(28) := "Slope Alarm 1 receive by CAN";
  gc_DbmTranslation_fr_Text616 : WSTRING(28) := "Slope Alarm 2 receive by CAN";
  gc_DbmTranslation_fr_Text617 : WSTRING(48) := "Slope Long Angle value with calibration offset 2";
  gc_DbmTranslation_fr_Text618 : WSTRING(49) := "Slope Trans Angle value with calibration offset 2";
  gc_DbmTranslation_fr_Text619 : WSTRING(51) := "Error code form emergency message encodeur turret 1";
  gc_DbmTranslation_fr_Text620 : WSTRING(55) := "Error register form emergency message encodeur turret 1";
  gc_DbmTranslation_fr_Text621 : WSTRING(51) := "Error code form emergency message encodeur turret 2";
  gc_DbmTranslation_fr_Text622 : WSTRING(55) := "Error register form emergency message encodeur turret 2";
  gc_DbmTranslation_fr_Text623 : WSTRING(46) := "Error code form emergency message mast measure";
  gc_DbmTranslation_fr_Text624 : WSTRING(50) := "Error register form emergency message mast measure";
  gc_DbmTranslation_fr_Text625 : WSTRING(41) := "State heart beat encodeur turret sensor 2";
  gc_DbmTranslation_fr_Text626 : WSTRING(46) := "Timeout Sdo Request Detected Encodeur Turret 1";
  gc_DbmTranslation_fr_Text627 : WSTRING(46) := "Timeout Sdo Request Detected Encodeur Turret 2";
  gc_DbmTranslation_fr_Text628 : WSTRING(31) := "Encodeur turret calibrate value";
  gc_DbmTranslation_fr_Text629 : WSTRING(33) := "Encodeur turret calibrate value 2";
  gc_DbmTranslation_fr_Text630 : WSTRING(29) := "User Log in Status (1=log in)";
  gc_DbmTranslation_fr_Text631 : WSTRING(21) := "Movement Allow Status";
  gc_DbmTranslation_fr_Text632 : WSTRING(20) := "Break Parking Status";
  gc_DbmTranslation_fr_Text633 : WSTRING(21) := "Break Faillure Status";
  gc_DbmTranslation_fr_Text634 : WSTRING(23) := "Turret Sector in Center";
  gc_DbmTranslation_fr_Text635 : WSTRING(23) := "Turret Sector in Center";
  gc_DbmTranslation_fr_Text636 : WSTRING(37) := "Vehicule in Train Mode (Speed in MPH)";
  gc_DbmTranslation_fr_Text637 : WSTRING(55) := "Incoherence between Lateral Stop and Key selector (A47)";
  gc_DbmTranslation_fr_Text638 : WSTRING(44) := "0=Work Mode activate 1=Site Acces Mode  (A4)";
  gc_DbmTranslation_fr_Text639 : WSTRING(35) := "Safety Electric Pump Activate (A44)";
  gc_DbmTranslation_fr_Text640 : WSTRING(38) := "Downhill between 150mm and 200mm (A13)";
  gc_DbmTranslation_fr_Text641 : WSTRING(22) := "Train Mode Allow (A10)";
  gc_DbmTranslation_fr_Text642 : WSTRING(34) := "Brake test need to be launch (A22)";
  gc_DbmTranslation_fr_Text643 : WSTRING(26) := "Brake Pressure Fault (A14)";
  gc_DbmTranslation_fr_Text644 : WSTRING(29) := "Activate Measuring Mast (A21)";
  gc_DbmTranslation_fr_Text645 : WSTRING(35) := "Auto Movement Direction Light (A23)";
  gc_DbmTranslation_fr_Text646 : WSTRING(38) := "Back Railway Axle in Low Position (A7)";
  gc_DbmTranslation_fr_Text647 : WSTRING(39) := "Front Railway Axle in Low Position (A7)";
  gc_DbmTranslation_fr_Text648 : WSTRING(37) := "Back Railway Axle Service Brake (A25)";
  gc_DbmTranslation_fr_Text649 : WSTRING(38) := "Front Railway Axle Service Brake (A25)";
  gc_DbmTranslation_fr_Text650 : WSTRING(34) := "Back Railway Axle Park Brake (A26)";
  gc_DbmTranslation_fr_Text651 : WSTRING(36) := "Front Railway Axle Park Brake (A26) ";
  gc_DbmTranslation_fr_Text652 : WSTRING(43) := "Status of Front Left Train Brake Test (A27)";
  gc_DbmTranslation_fr_Text653 : WSTRING(44) := "Status of Front Right Train Brake Test (A27)";
  gc_DbmTranslation_fr_Text654 : WSTRING(42) := "Status of Back Left Train Brake Test (A27)";
  gc_DbmTranslation_fr_Text655 : WSTRING(42) := "Status of Back Left Train Brake Test (A27)";
  gc_DbmTranslation_fr_Text656 : WSTRING(23) := "Status of the ARU alarm";
  gc_DbmTranslation_fr_Text657 : WSTRING(23) := "Engine use time in hour";
  gc_DbmTranslation_fr_Text658 : WSTRING(10) := "Engine RPM";
  gc_DbmTranslation_fr_Text659 : WSTRING(28) := "Vehicule Speed in Km/h * 100";
  gc_DbmTranslation_fr_Text660 : WSTRING(72) := "Lateralization Stop 1=bi lateralization 2=ALO Work 3=Multiple track (A3)";
  gc_DbmTranslation_fr_Text661 : WSTRING(64) := "Key Selector 1=bi lateralization 2=ALO Work 3=Multiple track(A6)";
  gc_DbmTranslation_fr_Text662 : WSTRING(38) := "Front Speed Railway Axle in Km/h (A24)";
  gc_DbmTranslation_fr_Text663 : WSTRING(31) := "Back Speed Railway Axle in Km/h";
  gc_DbmTranslation_fr_Text664 : WSTRING(59) := "Button for the calibration of the turret encoder is pressed";
  gc_DbmTranslation_fr_Text665 : WSTRING(47) := "Status of off track variable on test brake page";
  gc_DbmTranslation_fr_Text666 : WSTRING(51) := "Status of off track variable on run in process page";
  gc_DbmTranslation_fr_Text667 : WSTRING(41) := "Request status of osci service test brake";
  gc_DbmTranslation_fr_Text668 : WSTRING(42) := "Request status of fixed service test brake";
  gc_DbmTranslation_fr_Text669 : WSTRING(41) := "Request status of both service test brake";
  gc_DbmTranslation_fr_Text670 : WSTRING(38) := "Request status of osci park test brake";
  gc_DbmTranslation_fr_Text671 : WSTRING(39) := "Request status of fixed park test brake";
  gc_DbmTranslation_fr_Text672 : WSTRING(38) := "Request status of both park test brake";
  gc_DbmTranslation_fr_Text673 : WSTRING(43) := "Request status of osci service run in brake";
  gc_DbmTranslation_fr_Text674 : WSTRING(49) := "Request status of fixed service run in test brake";
  gc_DbmTranslation_fr_Text675 : WSTRING(48) := "Request status of both service run in test brake";
  gc_DbmTranslation_fr_Text676 : WSTRING(35) := "Test brake page is active on screen";
  gc_DbmTranslation_fr_Text677 : WSTRING(39) := "break in brake page is active on screen";
  gc_DbmTranslation_fr_Text678 : WSTRING(13) := "Serial Number";
  gc_DbmTranslation_fr_Text679 : WSTRING(18) := "BP Basket Validate";
  gc_DbmTranslation_fr_Text680 : WSTRING(19) := "Key Filter Overload";
  gc_DbmTranslation_fr_Text681 : WSTRING(13) := "Key Next Mode";
  gc_DbmTranslation_fr_Text682 : WSTRING(13) := "Key Prev Mode";
  gc_DbmTranslation_fr_Text683 : WSTRING(17) := "Key Signal Danger";
  gc_DbmTranslation_fr_Text684 : WSTRING(18) := "Key Flash Light ON";
  gc_DbmTranslation_fr_Text685 : WSTRING(18) := "Key Calib Mast Min";
  gc_DbmTranslation_fr_Text686 : WSTRING(18) := "Key Calib Mast Max";
  gc_DbmTranslation_fr_Text687 : WSTRING(17) := "KeyCalibMastValid";
  gc_DbmTranslation_fr_Text688 : WSTRING(24) := "Key Generator Activation";
  gc_DbmTranslation_fr_Text689 : WSTRING(40) := "raz distance travaled mast mesure button";
  gc_DbmTranslation_fr_Text690 : WSTRING(22) := "Key white lights 15746";
  gc_DbmTranslation_fr_Text691 : WSTRING(26) := "Osci 2nd Park Brake Select";
  gc_DbmTranslation_fr_Text692 : WSTRING(26) := "Fixe 2nd Park Brake Select";
  gc_DbmTranslation_fr_Text693 : WSTRING(18) := "RAZ controller Key";
  gc_DbmTranslation_fr_Text694 : WSTRING(29) := "Turret post selector input C1";
  gc_DbmTranslation_fr_Text695 : WSTRING(28) := "Radio Post Selector input C1";
  gc_DbmTranslation_fr_Text696 : WSTRING(30) := "Nacelle Post Selector input C1";
  gc_DbmTranslation_fr_Text697 : WSTRING(25) := "Up axle oscillant command";
  gc_DbmTranslation_fr_Text698 : WSTRING(27) := "Down axle oscillant command";
  gc_DbmTranslation_fr_Text699 : WSTRING(20) := "Up axle Fixe command";
  gc_DbmTranslation_fr_Text700 : WSTRING(21) := "Down axle Fixecommand";
  gc_DbmTranslation_fr_Text701 : WSTRING(27) := "Regime motor alternator rpm";
  gc_DbmTranslation_fr_Text702 : WSTRING(26) := "Entry telescope fdc sensor";
  gc_DbmTranslation_fr_Text703 : WSTRING(23) := "DElta arm folded sensor";
  gc_DbmTranslation_fr_Text704 : WSTRING(23) := "Booom Arm folded sensor";
  gc_DbmTranslation_fr_Text705 : WSTRING(23) := "Delta ram in lower zone";
  gc_DbmTranslation_fr_Text706 : WSTRING(30) := "Arrow arm angular sensor value";
  gc_DbmTranslation_fr_Text707 : WSTRING(33) := "Turret is in the rear center zone";
  gc_DbmTranslation_fr_Text708 : WSTRING(34) := "Turret is in the front center zone";
  gc_DbmTranslation_fr_Text709 : WSTRING(47) := "Folded delta arm zone detect with analog sensor";
  gc_DbmTranslation_fr_Text710 : WSTRING(47) := "Folded arrow arm zone detect with analog sensor";
  gc_DbmTranslation_fr_Text711 : WSTRING(21) := "No movement is during";
  gc_DbmTranslation_fr_Text712 : WSTRING(30) := "Delta arm angular sensor value";
  gc_DbmTranslation_fr_Text713 : WSTRING(31) := "Folded position of mast measure";
  gc_DbmTranslation_fr_Text714 : WSTRING(22) := "Transmission1 Pressure";
  gc_DbmTranslation_fr_Text715 : WSTRING(22) := "Transmission2 Pressure";
  gc_DbmTranslation_fr_Text716 : WSTRING(17) := "Active Help state";
  gc_DbmTranslation_fr_Text717 : WSTRING(25) := "Basket un center position";
  gc_DbmTranslation_fr_Text718 : WSTRING(31) := "Stop all movements Nacelle post";
  gc_DbmTranslation_fr_Text719 : WSTRING(39) := "Encodeur Mast measure value in centimer";
  gc_DbmTranslation_fr_Text720 : WSTRING(41) := "Flag when mast measure function is active";
  gc_DbmTranslation_fr_Text721 : WSTRING(34) := "Out of range transmission pressure";
  gc_DbmTranslation_fr_Text722 : WSTRING(21) := "Commande du gyrophare";
  gc_DbmTranslation_fr_Text723 : WSTRING(13) := "Moteur allumé";
  gc_DbmTranslation_fr_Text724 : WSTRING(27) := "Alarme du capteur téléscope";
  gc_DbmTranslation_fr_Text725 : WSTRING(30) := "Alarme sur le capteur tourelle";
  gc_DbmTranslation_fr_Text726 : WSTRING(26) := "Option White Light EN15746";
  gc_DbmTranslation_fr_Text727 : WSTRING(15) := "Safe man system";
  gc_DbmTranslation_fr_Text728 : WSTRING(18) := "Slope Mode from C1";
  gc_DbmTranslation_fr_Text729 : WSTRING(25) := "Cold Oil Tank Temperature";
  gc_DbmTranslation_fr_Text730 : WSTRING(24) := "Electric Motor Forbidden";
  gc_DbmTranslation_fr_Text731 : WSTRING(19) := "Rpm Electric Motor ";
  gc_DbmTranslation_fr_Text732 : WSTRING(21) := "Oil Tank Temperature ";
  gc_DbmTranslation_fr_Text733 : WSTRING(21) := "SOC stop regeneration";
  gc_DbmTranslation_fr_Text734 : WSTRING(12) := "Generator ON";
  gc_DbmTranslation_fr_Text735 : WSTRING(36) := "Active EV deviator movements command";
  gc_DbmTranslation_fr_Text736 : WSTRING(23) := "Test electrical from C1";
  gc_DbmTranslation_fr_Text737 : WSTRING(23) := "Automatic Mode Activate";
  gc_DbmTranslation_fr_Text738 : WSTRING(21) := "Silence Mode Activate";
  gc_DbmTranslation_fr_Text739 : WSTRING(30) := "Forcing Regeneration low level";
  gc_DbmTranslation_fr_Text740 : WSTRING(31) := "Forcing Regeneration High level";
  gc_DbmTranslation_fr_Text741 : WSTRING(17) := "EV Bypass command";
  gc_DbmTranslation_fr_Text742 : WSTRING(21) := "Motor speed CMD J1939";
  gc_DbmTranslation_fr_Text743 : WSTRING(50) := "Command to perform the calibration of turret angle";
  gc_DbmTranslation_fr_Text744 : WSTRING(64) := "Command to perform the calibration of turret angle intermediaire";
  gc_DbmTranslation_fr_Text745 : WSTRING(53) := "Command to perform the calibration of longetude angle";
  gc_DbmTranslation_fr_Text746 : WSTRING(55) := "Command to perform the calibration of transversal angle";
  gc_DbmTranslation_fr_Text747 : WSTRING(49) := "Command to saved calibration list value on EEPROM";
  gc_DbmTranslation_fr_Text748 : WSTRING(52) := "Acces chantier speed aplly to consigne max EvForward";
  gc_DbmTranslation_fr_Text749 : WSTRING(42) := "High speed aplly to consigne max EvForward";
  gc_DbmTranslation_fr_Text750 : WSTRING(41) := "Low speed aplly to consigne max EvForward";
  gc_DbmTranslation_fr_Text751 : WSTRING(67) := "Low speed apply to consigne max EvForward when test brake is needed";
  gc_DbmTranslation_fr_Text752 : WSTRING(55) := "Treshold slope vehicule angle for high speed (absolute)";
  gc_DbmTranslation_fr_Text753 : WSTRING(72) := "Hysteresis applied on the slope vehicule angle for high speed (relative)";
  gc_DbmTranslation_fr_Text754 : WSTRING(54) := "Treshold slope vehicule angle for low speed (absolute)";
  gc_DbmTranslation_fr_Text755 : WSTRING(71) := "Hysteresis applied on the slope vehicule angle for low speed (relative)";
  gc_DbmTranslation_fr_Text756 : WSTRING(93) := "Treshold angle of turret for low speed in (relative to TurretRear PosFront and NegFront zone)";
  gc_DbmTranslation_fr_Text757 : WSTRING(64) := "Hysteresis applied on the Treshold angle of turret for low speed";
  gc_DbmTranslation_fr_Text758 : WSTRING(34) := "Rear center position of the turret";
  gc_DbmTranslation_fr_Text759 : WSTRING(61) := "Front center position of the turret in the positive direction";
  gc_DbmTranslation_fr_Text760 : WSTRING(61) := "Front center position of the turret in the negative direction";
  gc_DbmTranslation_fr_Text761 : WSTRING(65) := "Limit speed on mode acces site speed wich trigger emergency brake";
  gc_DbmTranslation_fr_Text762 : WSTRING(58) := "Limit speed on mode highSpeed wich trigger emergency brake";
  gc_DbmTranslation_fr_Text763 : WSTRING(63) := "Limit speed on mode lowSpeed speed wich trigger emergency brake";
  gc_DbmTranslation_fr_Text764 : WSTRING(69) := "Limit speed on mode Low Speed Brake Test wich trigger emergency brake";
  gc_DbmTranslation_fr_Text765 : WSTRING(52) := "Acces chantier speed aplly to consigne max Backward ";
  gc_DbmTranslation_fr_Text766 : WSTRING(42) := "High speed aplly to consigne max Backward ";
  gc_DbmTranslation_fr_Text767 : WSTRING(41) := "Low speed aplly to consigne max Backward ";
  gc_DbmTranslation_fr_Text768 : WSTRING(68) := "Low speed apply to consigne max EvBackward when test brake is needed";
  gc_DbmTranslation_fr_Text769 : WSTRING(49) := "Test brake speed apply to consinge max Ev forward";
  gc_DbmTranslation_fr_Text770 : WSTRING(50) := "Test brake speed apply to consinge max Ev backward";
  gc_DbmTranslation_fr_Text771 : WSTRING(53) := "Break in brake speed apply to consinge max Ev forward";
  gc_DbmTranslation_fr_Text772 : WSTRING(54) := "Break in brake speed apply to consinge max Ev backward";
  gc_DbmTranslation_fr_Text773 : WSTRING(25) := "Arm speed rail hysteresis";
  gc_DbmTranslation_fr_Text774 : WSTRING(36) := "Arm low sector basket fault treshold";
  gc_DbmTranslation_fr_Text775 : WSTRING(26) := "Arm low zone for low speed";
  gc_DbmTranslation_fr_Text776 : WSTRING(38) := "Turret rear negatif low speed treshold";
  gc_DbmTranslation_fr_Text777 : WSTRING(38) := "Turret rear positif low speed treshold";
  gc_DbmTranslation_fr_Text778 : WSTRING(33) := "Slope thres of 2 deg for STRUKTON";
  gc_DbmTranslation_fr_Text779 : WSTRING(33) := "Slope thres of 4 deg for STRUKTON";
  gc_DbmTranslation_fr_Text780 : WSTRING(33) := "Slope thres of 6 deg for STRUKTON";
  gc_DbmTranslation_fr_Text781 : WSTRING(38) := "Slope Hyst for measure of slope angle ";
  gc_DbmTranslation_fr_Text782 : WSTRING(51) := "Turret Hyst for sector of turret versus slope angle";
  gc_DbmTranslation_fr_Text783 : WSTRING(41) := "Turret Sector for Slope angle below 2 Deg";
  gc_DbmTranslation_fr_Text784 : WSTRING(62) := "Turret Sector for Slope angle below 2 Deg with rotation basket";
  gc_DbmTranslation_fr_Text785 : WSTRING(41) := "Turret Sector for Slope angle below 4 Deg";
  gc_DbmTranslation_fr_Text786 : WSTRING(62) := "Turret Sector for Slope angle below 4 Deg with rotation basket";
  gc_DbmTranslation_fr_Text787 : WSTRING(41) := "Turret Sector for Slope angle below 6 Deg";
  gc_DbmTranslation_fr_Text788 : WSTRING(62) := "Turret Sector for Slope angle below 6 Deg with rotation basket";
  gc_DbmTranslation_fr_Text789 : WSTRING(60) := "Parameters to Prevention for Limit Speed in Acces Site Speed";
  gc_DbmTranslation_fr_Text790 : WSTRING(54) := "Parameters to Prevention for Limit Speed in High Speed";
  gc_DbmTranslation_fr_Text791 : WSTRING(53) := "Parameters to Prevention for Limit Speed in Low Speed";
  gc_DbmTranslation_fr_Text792 : WSTRING(58) := "Parameters to Prevention for Speed in Low Speed Brake Test";
  gc_DbmTranslation_fr_Text793 : WSTRING(76) := "Slope is over at high speed treshold (a hysteris is applied on the treshold)";
  gc_DbmTranslation_fr_Text794 : WSTRING(76) := "Slope is lower at low speed treshold (a hysteris is applied on the treshold)";
  gc_DbmTranslation_fr_Text795 : WSTRING(35) := "Turret angle in low speed rear zone";
  gc_DbmTranslation_fr_Text796 : WSTRING(44) := "Turret angle in low speed postiif front zone";
  gc_DbmTranslation_fr_Text797 : WSTRING(44) := "Turret angle in low speed negatif front zone";
  gc_DbmTranslation_fr_Text798 : WSTRING(30) := "Turret angle in low speed zone";
  gc_DbmTranslation_fr_Text799 : WSTRING(80) := "Enable simulation mode (use the simulation variables instead of the real inputs)";
  gc_DbmTranslation_fr_Text800 : WSTRING(0) := "";
  gc_DbmTranslation_fr_Text801 : WSTRING(0) := "";
  gc_DbmTranslation_fr_Text802 : WSTRING(0) := "";
  gc_DbmTranslation_fr_Text803 : WSTRING(0) := "";
  gc_DbmTranslation_fr_Text804 : WSTRING(0) := "";
  gc_DbmTranslation_fr_Text805 : WSTRING(0) := "";
  gc_DbmTranslation_fr_Text806 : WSTRING(0) := "";
  gc_DbmTranslation_fr_Text807 : WSTRING(0) := "";
  gc_DbmTranslation_fr_Text808 : WSTRING(0) := "";
  gc_DbmTranslation_fr_Text809 : WSTRING(0) := "";
  gc_DbmTranslation_fr_Text810 : WSTRING(0) := "";
  gc_DbmTranslation_fr_Text811 : WSTRING(0) := "";
  gc_DbmTranslation_fr_Text812 : WSTRING(0) := "";
  gc_DbmTranslation_fr_Text813 : WSTRING(0) := "";
  gc_DbmTranslation_fr_Text814 : WSTRING(0) := "";
  gc_DbmTranslation_fr_Text815 : WSTRING(0) := "";
  gc_DbmTranslation_fr_Text816 : WSTRING(0) := "";
  gc_DbmTranslation_fr_Text817 : WSTRING(0) := "";
  gc_DbmTranslation_fr_Text818 : WSTRING(0) := "";
  gc_DbmTranslation_fr_Text819 : WSTRING(49) := "Flag to detect exceeded of limit speed acces site";
  gc_DbmTranslation_fr_Text820 : WSTRING(43) := "Flag to detect exceeded of limit speed high";
  gc_DbmTranslation_fr_Text821 : WSTRING(48) := "Flag to detect exceeded of limit speed low speed";
  gc_DbmTranslation_fr_Text822 : WSTRING(55) := "Flag to detect exceeded of limit speed speed brake test";
  gc_DbmTranslation_fr_Text823 : WSTRING(32) := "Flag when one Litmit is exceeded";
  gc_DbmTranslation_fr_Text824 : WSTRING(21) := "Kinematic train allow";
  gc_DbmTranslation_fr_Text825 : WSTRING(31) := "Case of Slope angle below 2 deg";
  gc_DbmTranslation_fr_Text826 : WSTRING(31) := "Case of Slope angle below 4 deg";
  gc_DbmTranslation_fr_Text827 : WSTRING(31) := "Case of Slope angle below 6 deg";
  gc_DbmTranslation_fr_Text828 : WSTRING(37) := "Case of Slope angle higher than 6 deg";
  gc_DbmTranslation_fr_Text829 : WSTRING(36) := "Turret in Low Speed zone below 2 deg";
  gc_DbmTranslation_fr_Text830 : WSTRING(36) := "Turret in Low Speed zone below 4 deg";
  gc_DbmTranslation_fr_Text831 : WSTRING(36) := "Turret in Low Speed zone below 6 deg";
  gc_DbmTranslation_fr_Text832 : WSTRING(57) := "Turret in Low Speed zone below 2 deg with basket rotation";
  gc_DbmTranslation_fr_Text833 : WSTRING(57) := "Turret in Low Speed zone below 4 deg with basket rotation";
  gc_DbmTranslation_fr_Text834 : WSTRING(57) := "Turret in Low Speed zone below 6 deg with basket rotation";
  gc_DbmTranslation_fr_Text835 : WSTRING(43) := "Prevention for Limit Speed Acces Site Speed";
  gc_DbmTranslation_fr_Text836 : WSTRING(37) := "Prevention for Limit Speed High Speed";
  gc_DbmTranslation_fr_Text837 : WSTRING(36) := "Prevention for Limit Speed Low Speed";
  gc_DbmTranslation_fr_Text838 : WSTRING(41) := "Prevention for Limit Low Speed Brake Test";
  gc_DbmTranslation_fr_Text839 : WSTRING(35) := "Prevention exceeding of limit speed";
  gc_DbmTranslation_fr_Text840 : WSTRING(54) := "Authorize global low speed in add performance function";
  gc_DbmTranslation_fr_Text841 : WSTRING(51) := "N cycles brake need to make a validation brake test";
  gc_DbmTranslation_fr_Text842 : WSTRING(40) := "N cycles critical , limit speed to 3km/h";
  gc_DbmTranslation_fr_Text843 : WSTRING(44) := "Speed mini treshold to increment brake cycle";
  gc_DbmTranslation_fr_Text844 : WSTRING(41) := "Pressure treshold for osci service brake ";
  gc_DbmTranslation_fr_Text845 : WSTRING(41) := "Pressure treshold for fixe service brake ";
  gc_DbmTranslation_fr_Text846 : WSTRING(40) := "Pressure treshold for osci parking brake";
  gc_DbmTranslation_fr_Text847 : WSTRING(40) := "Pressure treshold for fixe parking brake";
  gc_DbmTranslation_fr_Text848 : WSTRING(38) := "Time for osci service brake valid test";
  gc_DbmTranslation_fr_Text849 : WSTRING(38) := "Time for fixe service brake valid test";
  gc_DbmTranslation_fr_Text850 : WSTRING(38) := "Time for osci parking brake valid test";
  gc_DbmTranslation_fr_Text851 : WSTRING(38) := "Time for fixe parking brake valid test";
  gc_DbmTranslation_fr_Text852 : WSTRING(33) := "Speed mini to brake automatically";
  gc_DbmTranslation_fr_Text853 : WSTRING(41) := "Valid condition to enable test brake time";
  gc_DbmTranslation_fr_Text854 : WSTRING(45) := "Number element of delta transmission pressure";
  gc_DbmTranslation_fr_Text855 : WSTRING(31) := "Seuil maximum de cycle de frein";
  gc_DbmTranslation_fr_Text856 : WSTRING(33) := "2nd Seuil de dépassement critique";
  gc_DbmTranslation_fr_Text857 : WSTRING(38) := "Temps pour la validation du test frein";
  gc_DbmTranslation_fr_Text858 : WSTRING(38) := "Temps pour la validation du test frein";
  gc_DbmTranslation_fr_Text859 : WSTRING(32) := "Threshold counter 2nd Park Brake";
  gc_DbmTranslation_fr_Text860 : WSTRING(39) := "Minimum Threshold Active 2nd Park Brake";
  gc_DbmTranslation_fr_Text861 : WSTRING(48) := "Fordid camera display when brake test is running";
  gc_DbmTranslation_fr_Text862 : WSTRING(24) := "Pressure efficiency rate";
  gc_DbmTranslation_fr_Text863 : WSTRING(34) := "Wich brake test selected on screen";
  gc_DbmTranslation_fr_Text864 : WSTRING(68) := "Flag when cycle brake perform is over parameters NCycleNeedBrakeTest";
  gc_DbmTranslation_fr_Text865 : WSTRING(67) := "Flag when cycle brake perform is over critial number of cycle brake";
  gc_DbmTranslation_fr_Text866 : WSTRING(19) := "Up position of axle";
  gc_DbmTranslation_fr_Text867 : WSTRING(21) := "Down position of axle";
  gc_DbmTranslation_fr_Text868 : WSTRING(58) := "Incoherence position axle and test mode in rail or offrail";
  gc_DbmTranslation_fr_Text869 : WSTRING(34) := "Test brake in rail or offrail mode";
  gc_DbmTranslation_fr_Text870 : WSTRING(28) := "Flag when brake test running";
  gc_DbmTranslation_fr_Text871 : WSTRING(34) := "Flag when valid brake test is done";
  gc_DbmTranslation_fr_Text872 : WSTRING(49) := "enable condition to increment cycke brake perform";
  gc_DbmTranslation_fr_Text873 : WSTRING(67) := "flag when a valid test brake is operared on oscillant service brake";
  gc_DbmTranslation_fr_Text874 : WSTRING(62) := "flag when a valid test brake is operared on fixe service brake";
  gc_DbmTranslation_fr_Text875 : WSTRING(67) := "flag when a valid test brake is operared on oscillant parking brake";
  gc_DbmTranslation_fr_Text876 : WSTRING(62) := "flag when a valid test brake is operared on fixe parking brake";
  gc_DbmTranslation_fr_Text877 : WSTRING(47) := "Simulation osci service breake select on screen";
  gc_DbmTranslation_fr_Text878 : WSTRING(47) := "Simulation fixe service breake select on screen";
  gc_DbmTranslation_fr_Text879 : WSTRING(47) := "Simulation osci parking breake select on screen";
  gc_DbmTranslation_fr_Text880 : WSTRING(47) := "Simulation fixe parking breake select on screen";
  gc_DbmTranslation_fr_Text881 : WSTRING(46) := "Simulation two service breake select on screen";
  gc_DbmTranslation_fr_Text882 : WSTRING(46) := "Simulation two parking breake select on screen";
  gc_DbmTranslation_fr_Text883 : WSTRING(39) := "Retain postition of joystick advanement";
  gc_DbmTranslation_fr_Text884 : WSTRING(38) := "Actual postion of joystick advancement";
  gc_DbmTranslation_fr_Text885 : WSTRING(29) := "Force oscillant service brake";
  gc_DbmTranslation_fr_Text886 : WSTRING(24) := "Force fixe service brake";
  gc_DbmTranslation_fr_Text887 : WSTRING(29) := "Force oscillant parking brake";
  gc_DbmTranslation_fr_Text888 : WSTRING(24) := "Force fixe parking brake";
  gc_DbmTranslation_fr_Text889 : WSTRING(35) := "stop all movement when a brake test";
  gc_DbmTranslation_fr_Text890 : WSTRING(94) := "Authorize translation rail when nacelle in transport mode and no incohrence with axle position";
  gc_DbmTranslation_fr_Text891 : WSTRING(38) := "Delta of transmission 1 and 2 preussre";
  gc_DbmTranslation_fr_Text892 : WSTRING(38) := "Valid condition enable test brake flag";
  gc_DbmTranslation_fr_Text893 : WSTRING(58) := "Flag when time out of valid condition to enable test brake";
  gc_DbmTranslation_fr_Text894 : WSTRING(20) := "Pourcent cycle brake";
  gc_DbmTranslation_fr_Text895 : WSTRING(18) := "Activation de l’EV";
  gc_DbmTranslation_fr_Text896 : WSTRING(18) := "Activation de l’EV";
  gc_DbmTranslation_fr_Text897 : WSTRING(76) := "Validation du test frein du frein de parc additionnel sur l’essieu Oscillant";
  gc_DbmTranslation_fr_Text898 : WSTRING(71) := "Validation du test frein du frein de parc additionnel sur l’essieu Fixe";
  gc_DbmTranslation_fr_Text899 : WSTRING(62) := "Variable de conversion du nombres de test frein en pourcentage";
  gc_DbmTranslation_fr_Text900 : WSTRING(46) := "Variable de dépassement du seuil de test frein";
  gc_DbmTranslation_fr_Text901 : WSTRING(55) := "Variable de dépassement du seuil critique de test frein";
  gc_DbmTranslation_fr_Text902 : WSTRING(29) := "Additionnal Park Brake Active";
  gc_DbmTranslation_fr_Text903 : WSTRING(30) := "Park Brake 2nd Pressure Active";
  gc_DbmTranslation_fr_Text904 : WSTRING(66) := "Minimum allowed turret angle for the consistency check in ALO mode";
  gc_DbmTranslation_fr_Text905 : WSTRING(66) := "Maximum allowed turret angle for the consistency check in ALO mode";
  gc_DbmTranslation_fr_Text906 : WSTRING(72) := "Minimum allowed turret angle for the consistency check in multilane mode";
  gc_DbmTranslation_fr_Text907 : WSTRING(72) := "Maximum allowed turret angle for the consistency check in multilane mode";
  gc_DbmTranslation_fr_Text908 : WSTRING(55) := "ALO mode - Rear zone threshold of the turret (absolute)";
  gc_DbmTranslation_fr_Text909 : WSTRING(81) := "ALO mode - Hysteresis applied on the rear zone threshold of the turret (relative)";
  gc_DbmTranslation_fr_Text910 : WSTRING(114) := "ALO mode - Threshold use to reduce speed before the rear zone of the turret (relative to the front zone threshold)";
  gc_DbmTranslation_fr_Text911 : WSTRING(56) := "ALO mode - Front zone threshold of the turret (absolute)";
  gc_DbmTranslation_fr_Text912 : WSTRING(82) := "ALO mode - Hysteresis applied on the front zone threshold of the turret (relative)";
  gc_DbmTranslation_fr_Text913 : WSTRING(115) := "ALO mode - Threshold use to reduce speed before the front zone of the turret (relative to the front zone threshold)";
  gc_DbmTranslation_fr_Text914 : WSTRING(66) := "ALO mode - Threshold of the lower zone of the arrow arm (absolute)";
  gc_DbmTranslation_fr_Text915 : WSTRING(85) := "ALO mode - Hysteresis applied on the lower zone threshold of the arrow arm (relative)";
  gc_DbmTranslation_fr_Text916 : WSTRING(118) := "ALO mode - Threshold use to reduce speed before the lower zone of the arrow arm (relative to the lower zone threshold)";
  gc_DbmTranslation_fr_Text917 : WSTRING(52) := "ALO mode - Turret rear end stop threshold (absolute)";
  gc_DbmTranslation_fr_Text918 : WSTRING(78) := "ALO mode - Hysteresis applied on the turret rear end stop threshold (relative)";
  gc_DbmTranslation_fr_Text919 : WSTRING(121) := "ALO mode - Threshold use to reduce speed before the rear end stop of the turret (relative to the rear end stop threshold)";
  gc_DbmTranslation_fr_Text920 : WSTRING(52) := "ALO mode - Turret rear end stop threshold (absolute)";
  gc_DbmTranslation_fr_Text921 : WSTRING(78) := "ALO mode - Hysteresis applied on the turret rear end stop threshold (relative)";
  gc_DbmTranslation_fr_Text922 : WSTRING(121) := "ALO mode - Threshold use to reduce speed before the rear end stop of the turret (relative to the rear end stop threshold)";
  gc_DbmTranslation_fr_Text923 : WSTRING(111) := "ALO mode - Threshold use to stop the turret before reaching the rear zone (relative to the rear zone threshold)";
  gc_DbmTranslation_fr_Text924 : WSTRING(86) := "ALO mode - Hysteresis applied to the rear zone stop threshold of the turret (relative)";
  gc_DbmTranslation_fr_Text925 : WSTRING(113) := "ALO mode - Threshold use to stop the turret before reaching the front zone (relative to the front zone threshold)";
  gc_DbmTranslation_fr_Text926 : WSTRING(87) := "ALO mode - Hysteresis applied to the front zone stop threshold of the turret (relative)";
  gc_DbmTranslation_fr_Text927 : WSTRING(116) := "ALO mode - Threshold use to stop the arrow arm before reaching the lower zone (relative to the lower zone threshold)";
  gc_DbmTranslation_fr_Text928 : WSTRING(90) := "ALO mode - Hysteresis applied to the lower zone stop threshold of the arrow arm (relative)";
  gc_DbmTranslation_fr_Text929 : WSTRING(34) := "Rail work mode selected by the key";
  gc_DbmTranslation_fr_Text930 : WSTRING(59) := "Consistency check - wrong turret abutment in bilateral mode";
  gc_DbmTranslation_fr_Text931 : WSTRING(59) := "Consistency check - wrong turret abutment in multilane mode";
  gc_DbmTranslation_fr_Text932 : WSTRING(53) := "Consistency check - wrong turret abutment in ALO mode";
  gc_DbmTranslation_fr_Text933 : WSTRING(77) := "Consistency check - wrong basket abutment in bilateral mode (only for France)";
  gc_DbmTranslation_fr_Text934 : WSTRING(77) := "Consistency check - wrong basket abutment in multilane mode (only for France)";
  gc_DbmTranslation_fr_Text935 : WSTRING(71) := "Consistency check - wrong basket abutment in ALO mode (only for France)";
  gc_DbmTranslation_fr_Text936 : WSTRING(43) := "Consistency check - wrong abutment detected";
  gc_DbmTranslation_fr_Text937 : WSTRING(59) := "Consistency check - wrong turret position in multilane mode";
  gc_DbmTranslation_fr_Text938 : WSTRING(59) := "Consistency check - wrong basket position in multilane mode";
  gc_DbmTranslation_fr_Text939 : WSTRING(53) := "Consistency check - wrong turret position in ALO mode";
  gc_DbmTranslation_fr_Text940 : WSTRING(43) := "Consistency check - wrong position detected";
  gc_DbmTranslation_fr_Text941 : WSTRING(49) := "Reduce the speed of the turret clockwise movement";
  gc_DbmTranslation_fr_Text942 : WSTRING(57) := "Reduce the speed of the turret counter clockwise movement";
  gc_DbmTranslation_fr_Text943 : WSTRING(47) := "Reduce the speed of the arrow arm down movement";
  gc_DbmTranslation_fr_Text944 : WSTRING(34) := "Stop the turret clockwise movement";
  gc_DbmTranslation_fr_Text945 : WSTRING(42) := "Stop the turret counter clockwise movement";
  gc_DbmTranslation_fr_Text946 : WSTRING(34) := "Stop the basket clockwise movement";
  gc_DbmTranslation_fr_Text947 : WSTRING(42) := "Stop the basket counter clockwise movement";
  gc_DbmTranslation_fr_Text948 : WSTRING(32) := "Stop the arrow arm down movement";
  gc_DbmTranslation_fr_Text949 : WSTRING(31) := "Stop the telescope out movement";
  gc_DbmTranslation_fr_Text950 : WSTRING(23) := "Turret in the rear zone";
  gc_DbmTranslation_fr_Text951 : WSTRING(24) := "Turret in the front zone";
  gc_DbmTranslation_fr_Text952 : WSTRING(27) := "Arrow arm in the lower zone";
  gc_DbmTranslation_fr_Text953 : WSTRING(60) := "Test variable for simulation - french version of the vehicle";
  gc_DbmTranslation_fr_Text954 : WSTRING(57) := "Test variable for simulation - basket abutment track side";
  gc_DbmTranslation_fr_Text955 : WSTRING(60) := "Test variable for simulation - basket abutment centered side";
  gc_DbmTranslation_fr_Text956 : WSTRING(54) := "Test variable for simulation - basket left side sensor";
  gc_DbmTranslation_fr_Text957 : WSTRING(55) := "Test variable for simulation - basket right side sensor";
  gc_DbmTranslation_fr_Text958 : WSTRING(49) := "Test variable for simulation - telescop in sensor";
  gc_DbmTranslation_fr_Text959 : WSTRING(54) := "Test variable for simulation - turret angular position";
  gc_DbmTranslation_fr_Text960 : WSTRING(57) := "Test variable for simulation - arrow arm angular position";
  gc_DbmTranslation_fr_Text961 : WSTRING(42) := "Abutment work mode selected by the sensors";
  gc_DbmTranslation_fr_Text962 : WSTRING(0) := "";
  gc_DbmTranslation_fr_Text963 : WSTRING(0) := "";
  gc_DbmTranslation_fr_Text964 : WSTRING(0) := "";
  gc_DbmTranslation_fr_Text965 : WSTRING(52) := "Delta arm treshold position for chenillard transport";
  gc_DbmTranslation_fr_Text966 : WSTRING(54) := "Delta arm hysteresis position for chenillard transport";
  gc_DbmTranslation_fr_Text967 : WSTRING(50) := "Arrow arm treshold position for off rail transport";
  gc_DbmTranslation_fr_Text968 : WSTRING(52) := "Arrow arm hysteresis position for off rail transport";
  gc_DbmTranslation_fr_Text969 : WSTRING(21) := "Turret angle thresold";
  gc_DbmTranslation_fr_Text970 : WSTRING(64) := "Bouton on screen to seleted the off rail mode for break in brake";
  gc_DbmTranslation_fr_Text971 : WSTRING(29) := "Force oscillant service brake";
  gc_DbmTranslation_fr_Text972 : WSTRING(24) := "Force fixe service brake";
  gc_DbmTranslation_fr_Text973 : WSTRING(29) := "Force oscillant parking brake";
  gc_DbmTranslation_fr_Text974 : WSTRING(24) := "Force fixe parking brake";
  gc_DbmTranslation_fr_Text975 : WSTRING(49) := "Stop all movement when a break in brake is during";
  gc_DbmTranslation_fr_Text976 : WSTRING(58) := "Incoherence position axle and test mode in rail or offrail";
  gc_DbmTranslation_fr_Text977 : WSTRING(53) := "Advancement period, reset every new advancement order";
  gc_DbmTranslation_fr_Text978 : WSTRING(22) := "Break in brake running";
  gc_DbmTranslation_fr_Text979 : WSTRING(47) := "Simu oscillant service brake selected on screen";
  gc_DbmTranslation_fr_Text980 : WSTRING(42) := "Simu fixe service brake selected on screen";
  gc_DbmTranslation_fr_Text981 : WSTRING(40) := "Simu 2 service brakes selected on screen";
  gc_DbmTranslation_fr_Text982 : WSTRING(47) := "Authorize transaltion on rail by break in brake";
  gc_DbmTranslation_fr_Text983 : WSTRING(32) := "Service brake selected on screen";
  gc_DbmTranslation_fr_Text984 : WSTRING(26) := "Advacnement period by 10ms";
  gc_DbmTranslation_fr_Text985 : WSTRING(30) := "Osci service brake in brake On";
  gc_DbmTranslation_fr_Text986 : WSTRING(30) := "Fixe service brake in brake On";
  gc_DbmTranslation_fr_Text987 : WSTRING(30) := "Both service brake in brake On";
  gc_DbmTranslation_fr_Text988 : WSTRING(36) := "Post selected to control the vehicle";
  gc_DbmTranslation_fr_Text989 : WSTRING(17) := "Enable the buzzer";
  gc_DbmTranslation_fr_Text990 : WSTRING(16) := "The slope is low";
  gc_DbmTranslation_fr_Text991 : WSTRING(17) := "The slope is high";
  gc_DbmTranslation_fr_Text992 : WSTRING(45) := "All commands of the nacelle post are disabled";
  gc_DbmTranslation_fr_Text993 : WSTRING(51) := "All commands of the radio command post are disabled";
  gc_DbmTranslation_fr_Text994 : WSTRING(44) := "All commands of the turret post are disabled";
  gc_DbmTranslation_fr_Text995 : WSTRING(41) := "Variable used to simulate the slope angle";
  gc_DbmTranslation_fr_Text996 : WSTRING(50) := "All ouput consigne of transaltion rail is disabled";
  gc_DbmTranslation_fr_Text997 : WSTRING(32) := "Authorise radio element position";
  gc_DbmTranslation_fr_Text998 : WSTRING(43) := "Threshold use to detect if the slope is low";
  gc_DbmTranslation_fr_Text999 : WSTRING(56) := "Hysteresis applied on the slope low threshold (relative)";
  gc_DbmTranslation_fr_Text1000 : WSTRING(44) := "Threshold use to detect if the slope is high";
  gc_DbmTranslation_fr_Text1001 : WSTRING(57) := "Hysteresis applied on the slope high threshold (relative)";
  gc_DbmTranslation_fr_Text1002 : WSTRING(26) := "Slope crawler max treshold";
  gc_DbmTranslation_fr_Text1003 : WSTRING(33) := "Life byte sent to the controllers";
  gc_DbmTranslation_fr_Text1004 : WSTRING(35) := "Delta arm move up button is pressed";
  gc_DbmTranslation_fr_Text1005 : WSTRING(37) := "Delta arm move down button is pressed";
  gc_DbmTranslation_fr_Text1006 : WSTRING(35) := "Arrow arm move up button is pressed";
  gc_DbmTranslation_fr_Text1007 : WSTRING(37) := "Arrow arm move down button is pressed";
  gc_DbmTranslation_fr_Text1008 : WSTRING(34) := "Pendular move up button is pressed";
  gc_DbmTranslation_fr_Text1009 : WSTRING(36) := "Pendular move down button is pressed";
  gc_DbmTranslation_fr_Text1010 : WSTRING(36) := "Telescope move out button is pressed";
  gc_DbmTranslation_fr_Text1011 : WSTRING(35) := "Telescope move in button is pressed";
  gc_DbmTranslation_fr_Text1012 : WSTRING(44) := "Basket inclinaison move up button is pressed";
  gc_DbmTranslation_fr_Text1013 : WSTRING(46) := "Basket inclinaison move down button is pressed";
  gc_DbmTranslation_fr_Text1014 : WSTRING(41) := "Rotate turret clockwise button is pressed";
  gc_DbmTranslation_fr_Text1015 : WSTRING(49) := "Rotate turret counter clockwise button is pressed";
  gc_DbmTranslation_fr_Text1016 : WSTRING(41) := "Basket rotation move up button is pressed";
  gc_DbmTranslation_fr_Text1017 : WSTRING(43) := "Basket rotation move down button is pressed";
  gc_DbmTranslation_fr_Text1018 : WSTRING(23) := "Key RPM Selection level";
  gc_DbmTranslation_fr_Text1019 : WSTRING(32) := "Key Desactivation RPM selection ";
  gc_DbmTranslation_fr_Text1020 : WSTRING(51) := "Activation forcing White Rail lights Front and Rear";
  gc_DbmTranslation_fr_Text1021 : WSTRING(16) := "Activation neons";
  gc_DbmTranslation_fr_Text1022 : WSTRING(19) := "Key Calibration Min";
  gc_DbmTranslation_fr_Text1023 : WSTRING(19) := "Key Calibration Max";
  gc_DbmTranslation_fr_Text1024 : WSTRING(26) := "Key Calibration Validation";
  gc_DbmTranslation_fr_Text1025 : WSTRING(89) := "Element choice 1=Telescope; 2=Arrow arm; 3=Delta arm; 4=Turret; 5=Slope; 6=Measuring Mast";
  gc_DbmTranslation_fr_Text1026 : WSTRING(27) := "Key Calibration Max (-180°)";
  gc_DbmTranslation_fr_Text1027 : WSTRING(28) := "Key Slope Longitudinal reset";
  gc_DbmTranslation_fr_Text1028 : WSTRING(27) := "Key Slope Transversal reset";
  gc_DbmTranslation_fr_Text1029 : WSTRING(76) := "DM_HIGH_HYDRAULIC_TEMP_CRAWLER - Overflow Threshold Fault Temperature Tracks";
  gc_DbmTranslation_fr_Text1030 : WSTRING(71) := "DM_HIGH_HYDRAULIC_TEMP_RAIL - Overflow Threshold Fault Temperature Rail";
  gc_DbmTranslation_fr_Text1031 : WSTRING(77) := "DM_ALARM_HYDRAULIC_TEMP_CRAWLER - Overflow Threshold Alarm Temperature Tracks";
  gc_DbmTranslation_fr_Text1032 : WSTRING(72) := "DM_ALARM_HYDRAULIC_TEMP_RAIL - Overflow Threshold Alarm Temperature Rail";
  gc_DbmTranslation_fr_Text1033 : WSTRING(69) := "DM_ONE_SPEED_SENSOR_FAULT - Tolerenace Threshold both 2 speed sensors";
  gc_DbmTranslation_fr_Text1034 : WSTRING(54) := "DM_SLOPE_FAULT - tolerance both 2 chanelles slope long";
  gc_DbmTranslation_fr_Text1035 : WSTRING(71) := "DM_OSCILLANT_CIRCUIT_FAULT - block isccilation axle pressure Threshold ";
  gc_DbmTranslation_fr_Text1036 : WSTRING(73) := "DM_OSCILLANT_CIRCUIT_FAULT - unblock isccilation axle pressure Threshold ";
  gc_DbmTranslation_fr_Text1037 : WSTRING(76) := "DM_SERVICE_BRAKE_PRESSURE_FAULT - Min service brake pressure fault threshold";
  gc_DbmTranslation_fr_Text1038 : WSTRING(76) := "DM_SERVICE_BRAKE_PRESSURE_FAULT - Max service brake pressure fault threshold";
  gc_DbmTranslation_fr_Text1039 : WSTRING(55) := "DM_SLOPE_FAULT  - tolerance both 2 chanelles slope long";
  gc_DbmTranslation_fr_Text1040 : WSTRING(79) := "DM_TRANS_CRAWLER_PRESSURE_HOOK - minimal pressure transmission when hook is off";
  gc_DbmTranslation_fr_Text1041 : WSTRING(80) := "DM_TURRET_SENSOR_FAULT  - tolerence trehsold betwen 2 channels of turrent sensor";
  gc_DbmTranslation_fr_Text1042 : WSTRING(108) := "DM_C0_OUT_OF_RANGE_JOY_DELTA_ARM_48XS - min alarm value of joytick delta arm in % according batterie voltage";
  gc_DbmTranslation_fr_Text1043 : WSTRING(108) := "DM_C0_OUT_OF_RANGE_JOY_DELTA_ARM_48XS - max alarm value of joytick delta arm in % according batterie voltage";
  gc_DbmTranslation_fr_Text1044 : WSTRING(108) := "DM_C0_OUT_OF_RANGE_JOY_ARROW_ARM_48XS - min alarm value of joytick arrow arm in % according batterie voltage";
  gc_DbmTranslation_fr_Text1045 : WSTRING(108) := "DM_C0_OUT_OF_RANGE_JOY_ARROW_ARM_48XS - max alarm value of joytick arrow arm in % according batterie voltage";
  gc_DbmTranslation_fr_Text1046 : WSTRING(116) := "DM_C0_OUT_OF_RANGE_JOY_TELESCOPE_ARM_48XS - min alarm value of joytick telescope arm in % according batterie voltage";
  gc_DbmTranslation_fr_Text1047 : WSTRING(116) := "DM_C0_OUT_OF_RANGE_JOY_TELESCOPE_ARM_48XS - max alarm value of joytick telescope arm in % according batterie voltage";
  gc_DbmTranslation_fr_Text1048 : WSTRING(123) := "DM_C0_OUT_OF_RANGE_JOY_ROT_TURRET_ARM_48XS - min alarm value of joytick rotation turret arm in % according batterie voltage";
  gc_DbmTranslation_fr_Text1049 : WSTRING(123) := "DM_C0_OUT_OF_RANGE_JOY_ROT_TURRET_ARM_48XS - max alarm value of joytick rotation turret arm in % according batterie voltage";
  gc_DbmTranslation_fr_Text1050 : WSTRING(120) := "DM_C0_OUT_OF_RANGE_JOY_ADVANCEMENT_48XS - min alarm value of joytick rotation turret arm in % according batterie voltage";
  gc_DbmTranslation_fr_Text1051 : WSTRING(120) := "DM_C0_OUT_OF_RANGE_JOY_ADVANCEMENT_48XS - max alarm value of joytick rotation turret arm in % according batterie voltage";
  gc_DbmTranslation_fr_Text1052 : WSTRING(61) := "DM_HIGH_HYDRAULIC_TEMP_RAIL - hysteresis treshold temperature";
  gc_DbmTranslation_fr_Text1053 : WSTRING(43) := "Reduce track speed when temperature default";
  gc_DbmTranslation_fr_Text1054 : WSTRING(82) := "Paramètre à ne jamais mettre à zéro. Utilisation pour le set du défaut de pression";
  gc_DbmTranslation_fr_Text1055 : WSTRING(32) := "Activation de l’alarme de bypass";
  gc_DbmTranslation_fr_Text1056 : WSTRING(17) := "Time Bypass Fault";
  gc_DbmTranslation_fr_Text1057 : WSTRING(48) := "Threshold of thermic transmission pressure Alarm";
  gc_DbmTranslation_fr_Text1058 : WSTRING(49) := "Threshold of electric transmission pressure Alarm";
  gc_DbmTranslation_fr_Text1059 : WSTRING(60) := "Time detect for the alarm of the Thermic pump on Translation";
  gc_DbmTranslation_fr_Text1060 : WSTRING(46) := "Time detect for the alarm of the Electric pump";
  gc_DbmTranslation_fr_Text1061 : WSTRING(0) := "";
  gc_DbmTranslation_fr_Text1062 : WSTRING(34) := "Fault on thermic pump transmission";
  gc_DbmTranslation_fr_Text1063 : WSTRING(55) := "Time to detect the fault on the thermic pump are passed";
  gc_DbmTranslation_fr_Text1064 : WSTRING(52) := "Active memorisation of the fault on the thermic pump";
  gc_DbmTranslation_fr_Text1065 : WSTRING(22) := "Fault on electric pump";
  gc_DbmTranslation_fr_Text1066 : WSTRING(56) := "Time to detect the fault on the electric pump are passed";
  gc_DbmTranslation_fr_Text1067 : WSTRING(57) := "Active memorisation of the fault on the DMC electric pump";
  gc_DbmTranslation_fr_Text1068 : WSTRING(40) := "Active fault on thermic or electric pump";
  gc_DbmTranslation_fr_Text1069 : WSTRING(0) := "";
  gc_DbmTranslation_fr_Text1070 : WSTRING(0) := "";
  gc_DbmTranslation_fr_Text1071 : WSTRING(0) := "";
  gc_DbmTranslation_fr_Text1072 : WSTRING(0) := "";
  gc_DbmTranslation_fr_Text1073 : WSTRING(0) := "";
  gc_DbmTranslation_fr_Text1074 : WSTRING(50) := "Last error code returned by the UART Init function";
  gc_DbmTranslation_fr_Text1075 : WSTRING(51) := "Last error code returned by the UART Write function";
  gc_DbmTranslation_fr_Text1076 : WSTRING(68) := "Successfully queued data butes (returned by the UART Write fucntion)";
  gc_DbmTranslation_fr_Text1077 : WSTRING(17) := "Displayed digit 1";
  gc_DbmTranslation_fr_Text1078 : WSTRING(17) := "Displayed digit 2";
  gc_DbmTranslation_fr_Text1079 : WSTRING(17) := "Displayed digit 3";
  gc_DbmTranslation_fr_Text1080 : WSTRING(17) := "Displayed digit 4";
  gc_DbmTranslation_fr_Text1081 : WSTRING(43) := "Data array given to the UART Write function";
  gc_DbmTranslation_fr_Text1082 : WSTRING(43) := "Data array given to the UART Write function";
  gc_DbmTranslation_fr_Text1083 : WSTRING(43) := "Data array given to the UART Write function";
  gc_DbmTranslation_fr_Text1084 : WSTRING(43) := "Data array given to the UART Write function";
  gc_DbmTranslation_fr_Text1085 : WSTRING(43) := "Data array given to the UART Write function";
  gc_DbmTranslation_fr_Text1086 : WSTRING(43) := "Data array given to the UART Write function";
  gc_DbmTranslation_fr_Text1087 : WSTRING(43) := "Data array given to the UART Write function";
  gc_DbmTranslation_fr_Text1088 : WSTRING(43) := "Data array given to the UART Write function";
  gc_DbmTranslation_fr_Text1089 : WSTRING(43) := "Data array given to the UART Write function";
  gc_DbmTranslation_fr_Text1090 : WSTRING(91) := "Refresh cycle time or the mast digital display ( cycle time of the message sent to display)";
  gc_DbmTranslation_fr_Text1091 : WSTRING(0) := "";
  gc_DbmTranslation_fr_Text1092 : WSTRING(0) := "";
  gc_DbmTranslation_fr_Text1093 : WSTRING(0) := "";
  gc_DbmTranslation_fr_Text1094 : WSTRING(0) := "";
  gc_DbmTranslation_fr_Text1095 : WSTRING(0) := "";
  gc_DbmTranslation_fr_Text1096 : WSTRING(0) := "";
  gc_DbmTranslation_fr_Text1097 : WSTRING(0) := "";
  gc_DbmTranslation_fr_Text1098 : WSTRING(0) := "";
  gc_DbmTranslation_fr_Text1099 : WSTRING(0) := "";
  gc_DbmTranslation_fr_Text1100 : WSTRING(0) := "";
  gc_DbmTranslation_fr_Text1101 : WSTRING(0) := "";
  gc_DbmTranslation_fr_Text1102 : WSTRING(0) := "";
  gc_DbmTranslation_fr_Text1103 : WSTRING(47) := "Autorisation of translation with unfolded arrow";
  gc_DbmTranslation_fr_Text1104 : WSTRING(43) := "Validation of Telescope sector to translate";
  gc_DbmTranslation_fr_Text1105 : WSTRING(49) := "Validation of First Telescope sector to translate";
  gc_DbmTranslation_fr_Text1106 : WSTRING(41) := "All Post interdict fot mast function SNCF";
  gc_DbmTranslation_fr_Text1107 : WSTRING(39) := "Interdiction of nacelle and turret post";
  gc_DbmTranslation_fr_Text1108 : WSTRING(36) := "SNCF contact mast in folded position";
  gc_DbmTranslation_fr_Text1109 : WSTRING(43) := "Maximum Pvg Translation Rail on Electric Av";
  gc_DbmTranslation_fr_Text1110 : WSTRING(43) := "Maximum Pvg Translation Rail on Electric Ar";
  gc_DbmTranslation_fr_Text1111 : WSTRING(43) := "Minimum Pvg Translation Rail on Electric Av";
  gc_DbmTranslation_fr_Text1112 : WSTRING(43) := "Minimum Pvg Translation Rail on Electric Ar";
  gc_DbmTranslation_fr_Text1113 : WSTRING(56) := "Translation on Rail with Electric Ramp Time Accelaration";
  gc_DbmTranslation_fr_Text1114 : WSTRING(56) := "Translation on Rail with Electric Ramp Time Deceleration";
  gc_DbmTranslation_fr_Text1115 : WSTRING(48) := "Translation on Rail with Electric Ramp Time Stop";
  gc_DbmTranslation_fr_Text1116 : WSTRING(30) := "Electric Pump Pressure Maximum";
  gc_DbmTranslation_fr_Text1117 : WSTRING(33) := "Electric Pump Pressure Hysteresys";
  gc_DbmTranslation_fr_Text1118 : WSTRING(39) := "Electric motor maximum Rpm Translation ";
  gc_DbmTranslation_fr_Text1119 : WSTRING(39) := "Electric motor minimum Rpm Translation ";
  gc_DbmTranslation_fr_Text1120 : WSTRING(56) := "Pourcent minimum for transaltion PVG on the high 50 side";
  gc_DbmTranslation_fr_Text1121 : WSTRING(55) := "Pourcent minimum for transaltion PVG on the low 50 side";
  gc_DbmTranslation_fr_Text1122 : WSTRING(38) := "Ramp time for the thermic regeneration";
  gc_DbmTranslation_fr_Text1123 : WSTRING(29) := "Pressure pump Regenration Max";
  gc_DbmTranslation_fr_Text1124 : WSTRING(32) := "Pressure pump Regeneration reset";
  gc_DbmTranslation_fr_Text1125 : WSTRING(34) := "Current reset regeneration thermic";
  gc_DbmTranslation_fr_Text1126 : WSTRING(52) := "Minimum current for the regeneration in thermic mode";
  gc_DbmTranslation_fr_Text1127 : WSTRING(52) := "Maximum current for the regeneration in thermic mode";
  gc_DbmTranslation_fr_Text1128 : WSTRING(53) := "Maximum current for the regeneration in electric mode";
  gc_DbmTranslation_fr_Text1129 : WSTRING(25) := "Low battery level for SOC";
  gc_DbmTranslation_fr_Text1130 : WSTRING(28) := "Minimum voltage Dc Converter";
  gc_DbmTranslation_fr_Text1131 : WSTRING(42) := "Number of fault cycle from de DC converter";
  gc_DbmTranslation_fr_Text1132 : WSTRING(32) := "RPM regeneration brake auto mode";
  gc_DbmTranslation_fr_Text1133 : WSTRING(35) := "Torque regeneration brake auto mode";
  gc_DbmTranslation_fr_Text1134 : WSTRING(32) := "RPM regeneration brake high mode";
  gc_DbmTranslation_fr_Text1135 : WSTRING(35) := "Torque regeneration brake high mode";
  gc_DbmTranslation_fr_Text1136 : WSTRING(29) := "Number of samples average Rpm";
  gc_DbmTranslation_fr_Text1137 : WSTRING(24) := "Regen Pump Pressure Hyst";
  gc_DbmTranslation_fr_Text1138 : WSTRING(38) := "Regen Brake Torque From Pressur Coef K";
  gc_DbmTranslation_fr_Text1139 : WSTRING(32) := "RegenBrakeTorqueFromPressurRange";
  gc_DbmTranslation_fr_Text1140 : WSTRING(42) := "Autorize Translation on Rail with Electric";
  gc_DbmTranslation_fr_Text1141 : WSTRING(46) := "Pvg Translation on Rail with Electric Consigne";
  gc_DbmTranslation_fr_Text1142 : WSTRING(31) := "Electric Pump Pressure Exceeded";
  gc_DbmTranslation_fr_Text1143 : WSTRING(42) := "Stop Ramp Pvg Translation on Rail Electric";
  gc_DbmTranslation_fr_Text1144 : WSTRING(41) := "Translation on Rail Electric Ramp Ongoing";
  gc_DbmTranslation_fr_Text1145 : WSTRING(42) := "Translation on Rail Thermique Ramp Ongoing";
  gc_DbmTranslation_fr_Text1146 : WSTRING(30) := "Rpm of Pvg Translation on Rail";
  gc_DbmTranslation_fr_Text1147 : WSTRING(39) := "Impossible reloaded baterry Pictogramme";
  gc_DbmTranslation_fr_Text1148 : WSTRING(17) := "Low level baterry";
  gc_DbmTranslation_fr_Text1149 : WSTRING(43) := "Electric pump pressure maximum regeneration";
  gc_DbmTranslation_fr_Text1150 : WSTRING(41) := "Electric pump pressure Reset regeneration";
  gc_DbmTranslation_fr_Text1151 : WSTRING(23) := "Autorize raz controller";
  gc_DbmTranslation_fr_Text1152 : WSTRING(29) := "Voltage Dc Converter in Fault";
  gc_DbmTranslation_fr_Text1153 : WSTRING(20) := "Battery Error Code 1";
  gc_DbmTranslation_fr_Text1154 : WSTRING(27) := "Picto Ask Resart Controller";
  gc_DbmTranslation_fr_Text1155 : WSTRING(23) := "Instant Current Battery";
  gc_DbmTranslation_fr_Text1156 : WSTRING(24) := "Instant Volatage Battery";
  gc_DbmTranslation_fr_Text1157 : WSTRING(17) := "load rate battery";
  gc_DbmTranslation_fr_Text1158 : WSTRING(29) := "Battery Power Reduction Ratio";
  gc_DbmTranslation_fr_Text1159 : WSTRING(32) := "Battery Recovery Reduction Ratio";
  gc_DbmTranslation_fr_Text1160 : WSTRING(20) := "Battery Error Code 1";
  gc_DbmTranslation_fr_Text1161 : WSTRING(21) := "Battery Error Value 1";
  gc_DbmTranslation_fr_Text1162 : WSTRING(31) := "Battery Regeneration Authorized";
  gc_DbmTranslation_fr_Text1163 : WSTRING(11) := "RPM request";
  gc_DbmTranslation_fr_Text1164 : WSTRING(38) := "Generator regeneration speed set point";
  gc_DbmTranslation_fr_Text1165 : WSTRING(44) := "Generator regeneration battery current limit";
  gc_DbmTranslation_fr_Text1166 : WSTRING(20) := "Forward Byte 6 Bit 0";
  gc_DbmTranslation_fr_Text1167 : WSTRING(21) := "Backward Byte 6 Bit 1";
  gc_DbmTranslation_fr_Text1168 : WSTRING(23) := "FootSwitch Byte 6 Bit 2";
  gc_DbmTranslation_fr_Text1169 : WSTRING(22) := "Interlock Byte 6 Bit 3";
  gc_DbmTranslation_fr_Text1170 : WSTRING(32) := "Regeneration Enable Byte 6 Bit 6";
  gc_DbmTranslation_fr_Text1171 : WSTRING(15) := "Roll over count";
  gc_DbmTranslation_fr_Text1172 : WSTRING(27) := "Drive battery current limit";
  gc_DbmTranslation_fr_Text1173 : WSTRING(34) := "Regeneration battery Current limit";
  gc_DbmTranslation_fr_Text1174 : WSTRING(11) := "Battery SOC";
  gc_DbmTranslation_fr_Text1175 : WSTRING(15) := "Roll over count";
  gc_DbmTranslation_fr_Text1176 : WSTRING(16) := "Actual speed RPM";
  gc_DbmTranslation_fr_Text1177 : WSTRING(15) := "Battery Current";
  gc_DbmTranslation_fr_Text1178 : WSTRING(15) := "Roll over count";
  gc_DbmTranslation_fr_Text1179 : WSTRING(10) := "Fault code";
  gc_DbmTranslation_fr_Text1180 : WSTRING(14) := "Fault sub code";
  gc_DbmTranslation_fr_Text1181 : WSTRING(13) := "Motor current";
  gc_DbmTranslation_fr_Text1182 : WSTRING(22) := "Drive status indicator";
  gc_DbmTranslation_fr_Text1183 : WSTRING(21) := "Speed limit indicator";
  gc_DbmTranslation_fr_Text1184 : WSTRING(13) := "Actual Torque";
  gc_DbmTranslation_fr_Text1185 : WSTRING(22) := "Torque limit Indicator";
  gc_DbmTranslation_fr_Text1186 : WSTRING(15) := "Roll over count";
  gc_DbmTranslation_fr_Text1187 : WSTRING(21) := "Controler Temperature";
  gc_DbmTranslation_fr_Text1188 : WSTRING(17) := "Motor Temperature";
  gc_DbmTranslation_fr_Text1189 : WSTRING(21) := "Motor limit indicator";
  gc_DbmTranslation_fr_Text1190 : WSTRING(15) := "Roll over count";
  gc_DbmTranslation_fr_Text1191 : WSTRING(15) := "Battery Voltage";
  gc_DbmTranslation_fr_Text1192 : WSTRING(27) := "Battery Discharge indicator";
  gc_DbmTranslation_fr_Text1193 : WSTRING(17) := "Waiting Heartbeat";
  gc_DbmTranslation_fr_Text1194 : WSTRING(21) := "TimeOut Dmc Heartbeat";
